KUKA KRL program: MyProgram_130().src

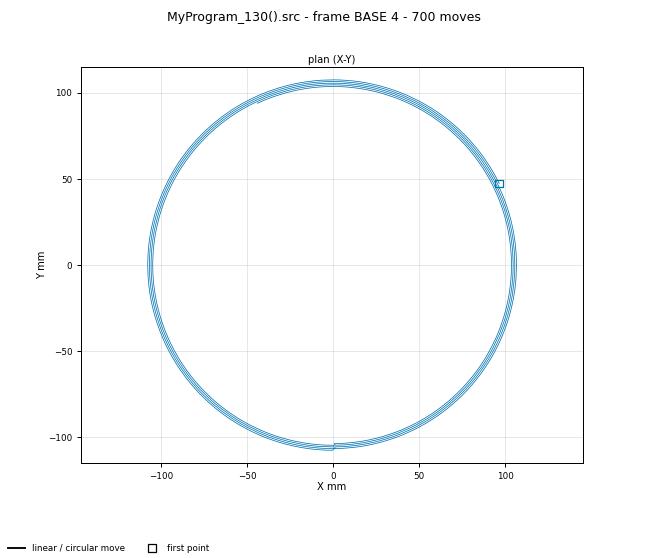
[picture p0: tool path of MyProgram_130().src in frame BASE 4, 700 of 700 moves have a stored position in this frame; points joined in program order, loops and branches not executed]
&ACCESS RVP
&REL 1
&PARAM TEMPLATE = C:\KRC\Roboter\Template\vorgabe
&PARAM EDITMASK = *
DEF MyProgram_130()
; ---- Setting reference (Base) ----
$BASE = BASE_DATA[4]

; --------------------------
; ---- Setting tool (TCP) ----
$TOOL = TOOL_DATA[3]
; --------------------------

$VEL.CP = VEL_APROX_PRINT
Startdeposition()
$VEL.CP = VEL_PRINT
LIN {X 96.6585,Y 47.3768,Z 107,A 22.2478,B 24.9305,C -1.9249,E1 25.1427,E2 423.328} C_DIS
LIN {X 94.8383,Y 50.9225,Z 107,A 24.2361,B 24.9305,C -1.9249,E1 25.1401,E2 421.3499} C_DIS
LIN {X 92.9821,Y 54.2393,Z 107,A 26.2737,B 24.9301,C -1.931,E1 25.1372,E2 419.3085} C_DIS
LIN {X 91.1089,Y 57.3278,Z 107,A 28.1051,B 24.9301,C -1.9322,E1 25.1346,E2 417.4838} C_DIS
LIN {X 89.1092,Y 60.3882,Z 107,A 30.0749,B 24.9296,C -1.9383,E1 25.1315,E2 415.5094} C_DIS
LIN {X 86.9613,Y 63.4425,Z 107,A 31.9479,B 24.9296,C -1.9383,E1 25.1285,E2 413.6455} C_DIS
LIN {X 84.9221,Y 66.1494,Z 107,A 33.8072,B 24.9291,C -1.9451,E1 25.1253,E2 411.779} C_DIS
LIN {X 82.7658,Y 68.826,Z 107,A 35.6176,B 24.9288,C -1.9486,E1 25.1221,E2 409.9685} C_DIS
LIN {X 79.7659,Y 72.2838,Z 107,A 38.1989,B 24.9279,C -1.9604,E1 25.1173,E2 407.3711} C_DIS
LIN {X 76.7784,Y 75.4477,Z 107,A 40.3094,B 24.9282,C -1.9567,E1 25.1132,E2 405.2784} C_DIS
LIN {X 74.3299,Y 77.8622,Z 107,A 42.0113,B 24.9283,C -1.955,E1 25.1098,E2 403.5875} C_DIS
LIN {X 71.8944,Y 80.1149,Z 107,A 43.9014,B 24.9277,C -1.9639,E1 25.1059,E2 401.684} C_DIS
LIN {X 69.2564,Y 82.4081,Z 107,A 45.8045,B 24.9273,C -1.9693,E1 25.1019,E2 399.7755} C_DIS
LIN {X 65.4421,Y 85.4672,Z 107,A 48.451,B 24.9268,C -1.976,E1 25.096,E2 397.1231} C_DIS
LIN {X 62.7263,Y 87.4795,Z 107,A 50.3374,B 24.9263,C -1.9828,E1 25.0918,E2 395.2272} C_DIS
LIN {X 59.7326,Y 89.5519,Z 107,A 52.0715,B 24.9267,C -1.9774,E1 25.0878,E2 393.5119} C_DIS
LIN {X 57.005,Y 91.3106,Z 107,A 53.7544,B 24.9267,C -1.9782,E1 25.0838,E2 391.8323} C_DIS
LIN {X 54.1931,Y 93.0092,Z 107,A 55.7988,B 24.9255,C -1.9932,E1 25.0788,E2 389.7588} C_DIS
LIN {X 50.2355,Y 95.2029,Z 107,A 57.8693,B 24.9263,C -1.9823,E1 25.0738,E2 387.7199} C_DIS
LIN {X 47.8532,Y 96.4223,Z 107,A 59.6078,B 24.9252,C -1.9973,E1 25.0694,E2 385.9507} C_DIS
LIN {X 43.6886,Y 98.3811,Z 107,A 61.7829,B 24.9259,C -1.9886,E1 25.064,E2 383.8015} C_DIS
LIN {X 40.8548,Y 99.59,Z 107,A 63.442,B 24.9257,C -1.9912,E1 25.0597,E2 382.1403} C_DIS
LIN {X 37.0788,Y 101.0564,Z 107,A 65.6254,B 24.9254,C -1.9944,E1 25.054,E2 379.9539} C_DIS
LIN {X 33.3917,Y 102.334,Z 107,A 67.6345,B 24.9254,C -1.9934,E1 25.0487,E2 377.9512} C_DIS
LIN {X 30.598,Y 103.2035,Z 107,A 69.2165,B 24.9254,C -1.9955,E1 25.0444,E2 376.3668} C_DIS
LIN {X 27.4751,Y 104.0802,Z 107,A 71.0057,B 24.9251,C -1.9992,E1 25.0396,E2 374.5718} C_DIS
LIN {X 24.1955,Y 104.8893,Z 107,A 72.6636,B 24.9254,C -1.9945,E1 25.0351,E2 372.9274} C_DIS
LIN {X 19.4871,Y 105.8661,Z 107,A 75.8484,B 24.9234,C -2.0212,E1 25.0262,E2 369.6832} C_DIS
LIN {X 15.5445,Y 106.5163,Z 107,A 77.4337,B 24.925,C -1.9997,E1 25.022,E2 368.1504} C_DIS
LIN {X 12.0252,Y 106.9712,Z 107,A 79.4475,B 24.9246,C -2.0051,E1 25.0164,E2 366.1252} C_DIS
LIN {X 8.1375,Y 107.3367,Z 107,A 81.5895,B 24.9244,C -2.0078,E1 25.0104,E2 363.9779} C_DIS
LIN {X 3.8187,Y 107.5773,Z 107,A 83.6882,B 24.925,C -1.9995,E1 25.0046,E2 361.8996} C_DIS
LIN {X 0.959,Y 107.64,Z 107,A 85.3969,B 24.9245,C -2.0067,E1 24.9998,E2 360.1738} C_DIS
LIN {X -6.6056,Y 107.443,Z 107,A 89.3666,B 24.9248,C -2.0031,E1 24.9887,E2 356.2122} C_DIS
LIN {X -10.3707,Y 107.1442,Z 107,A 92.1892,B 24.9224,C -2.0346,E1 24.9807,E2 353.313} C_DIS
LIN {X -15.902,Y 106.4642,Z 107,A 94.2252,B 24.9253,C -1.9955,E1 24.9753,E2 351.3684} C_DIS
LIN {X -19.0755,Y 105.9402,Z 107,A 95.8763,B 24.9256,C -1.9919,E1 24.9708,E2 349.7242} C_DIS
LIN {X -22.435,Y 105.2812,Z 107,A 97.6602,B 24.9258,C -1.9888,E1 24.9659,E2 347.9455} C_DIS
LIN {X -25.6012,Y 104.5551,Z 107,A 99.5013,B 24.9256,C -1.9916,E1 24.9609,E2 346.0953} C_DIS
LIN {X -28.8893,Y 103.6958,Z 107,A 101.1251,B 24.9263,C -1.9825,E1 24.9566,E2 344.4908} C_DIS
LIN {X -31.4867,Y 102.9366,Z 107,A 102.8288,B 24.9257,C -1.9912,E1 24.9519,E2 342.7635} C_DIS
LIN {X -37.5976,Y 100.8659,Z 107,A 106.2811,B 24.9259,C -1.9875,E1 24.9428,E2 339.3131} C_DIS
LIN {X -41.0114,Y 99.5262,Z 107,A 108.0603,B 24.9266,C -1.9781,E1 24.9383,E2 337.5524} C_DIS
LIN {X -44.3883,Y 98.0658,Z 107,A 110.1145,B 24.9266,C -1.979,E1 24.933,E2 335.4914} C_DIS
LIN {X -48.0689,Y 96.3154,Z 107,A 112.4048,B 24.9265,C -1.9802,E1 24.9272,E2 333.1923} C_DIS
LIN {X -50.9886,Y 94.8024,Z 107,A 114.0879,B 24.9269,C -1.9746,E1 24.9231,E2 331.5177} C_DIS
LIN {X -53.859,Y 93.2012,Z 107,A 115.8714,B 24.927,C -1.9728,E1 24.9188,E2 329.7331} C_DIS
LIN {X -56.3491,Y 91.7183,Z 107,A 117.5087,B 24.927,C -1.9736,E1 24.9149,E2 328.089} C_DIS
LIN {X -59.3917,Y 89.7766,Z 107,A 119.7982,B 24.9262,C -1.984,E1 24.9095,E2 325.7671} C_DIS
LIN {X -62.5149,Y 87.6303,Z 107,A 121.9673,B 24.9261,C -1.9858,E1 24.9045,E2 323.5863} C_DIS
LIN {X -66.0582,Y 84.9921,Z 107,A 123.752,B 24.928,C -1.9591,E1 24.9007,E2 321.8588} C_DIS
LIN {X -69.9051,Y 81.8561,Z 107,A 126.4305,B 24.9284,C -1.9546,E1 24.8949,E2 319.1806} C_DIS
LIN {X -73.3692,Y 78.7658,Z 107,A 129.2092,B 24.9279,C -1.9606,E1 24.8891,E2 316.3765} C_DIS
LIN {X -76.0308,Y 76.2023,Z 107,A 131.5737,B 24.9272,C -1.9709,E1 24.8844,E2 313.9773} C_DIS
LIN {X -79.385,Y 72.6996,Z 107,A 133.1703,B 24.9304,C -1.9272,E1 24.8816,E2 312.4779} C_DIS
LIN {X -83.0404,Y 68.4953,Z 107,A 136.283,B 24.9305,C -1.925,E1 24.8759,E2 309.3563} C_DIS
LIN {X -85.2435,Y 65.7323,Z 107,A 138.1744,B 24.9309,C -1.9204,E1 24.8726,E2 307.467} C_DIS
LIN {X -86.7483,Y 63.7335,Z 107,A 139.524,B 24.9311,C -1.9174,E1 24.8704,E2 306.1179} C_DIS
LIN {X -88.2223,Y 61.6774,Z 107,A 140.9553,B 24.9311,C -1.9169,E1 24.8681,E2 304.6809} C_DIS
LIN {X -89.7399,Y 59.4474,Z 107,A 142.4812,B 24.9311,C -1.9162,E1 24.8657,E2 303.1489} C_DIS
LIN {X -91.7156,Y 56.3535,Z 107,A 144.4514,B 24.9315,C -1.9113,E1 24.8628,E2 301.1806} C_DIS
LIN {X -93.6411,Y 53.0935,Z 107,A 146.4172,B 24.9321,C -1.9036,E1 24.86,E2 299.2228} C_DIS
LIN {X -95.5947,Y 49.4882,Z 107,A 148.929,B 24.9316,C -1.9094,E1 24.8567,E2 296.6836} C_DIS
LIN {X -98.2788,Y 43.9152,Z 107,A 151.9288,B 24.9331,C -1.8886,E1 24.8532,E2 293.7172} C_DIS
LIN {X -99.7804,Y 40.3869,Z 107,A 154.0677,B 24.9333,C -1.886,E1 24.8509,E2 291.5727} C_DIS
LIN {X -101.0566,Y 37.0783,Z 107,A 155.7378,B 24.9343,C -1.8721,E1 24.8493,E2 289.9264} C_DIS
LIN {X -102.2236,Y 33.733,Z 107,A 157.8972,B 24.934,C -1.8763,E1 24.8474,E2 287.7446} C_DIS
LIN {X -103.3972,Y 29.9431,Z 107,A 159.9805,B 24.9345,C -1.8686,E1 24.8457,E2 285.6677} C_DIS
LIN {X -104.3459,Y 26.4433,Z 107,A 162.0668,B 24.9345,C -1.8683,E1 24.8442,E2 283.57} C_DIS
LIN {X -105.411,Y 21.8113,Z 107,A 164.295,B 24.9359,C -1.849,E1 24.8429,E2 281.3746} C_DIS
LIN {X -105.8892,Y 19.3588,Z 107,A 165.5472,B 24.9364,C -1.8418,E1 24.8423,E2 280.1321} C_DIS
LIN {X -106.3948,Y 16.3507,Z 107,A 167.2943,B 24.9364,C -1.8412,E1 24.8415,E2 278.3761} C_DIS
LIN {X -106.8679,Y 12.907,Z 107,A 169.2441,B 24.9366,C -1.8389,E1 24.8408,E2 276.4202} C_DIS
LIN {X -107.1659,Y 10.1354,Z 107,A 171.2847,B 24.9355,C -1.8548,E1 24.8403,E2 274.3293} C_DIS
LIN {X -107.4711,Y 6.0983,Z 107,A 173.0589,B 24.937,C -1.8336,E1 24.84,E2 272.595} C_DIS
LIN {X -107.6446,Y 0.1321,Z 107,A 177.1432,B 24.9353,C -1.8574,E1 24.8398,E2 268.4294} C_DIS
LIN {X -107.4825,Y -5.891,Z 107,A 179.2876,B 24.9388,C -1.8072,E1 24.8401,E2 266.3918} C_DIS
LIN {X -107.2538,Y -9.1743,Z 107,A -178.835,B 24.9388,C -1.8062,E1 24.8405,E2 264.5055} C_DIS
LIN {X -106.9,Y -12.633,Z 107,A -177.0787,B 24.9395,C -1.7968,E1 24.8411,E2 262.761} C_DIS
LIN {X -106.404,Y -16.2911,Z 107,A -175.0871,B 24.9398,C -1.7916,E1 24.8418,E2 260.7701} C_DIS
LIN {X -105.8218,Y -19.7319,Z 107,A -173.144,B 24.94,C -1.7889,E1 24.8428,E2 258.8218} C_DIS
LIN {X -105.1397,Y -23.0837,Z 107,A -171.3092,B 24.9404,C -1.7838,E1 24.8439,E2 256.9885} C_DIS
LIN {X -104.3676,Y -26.3591,Z 107,A -169.601,B 24.9409,C -1.7751,E1 24.845,E2 255.2908} C_DIS
LIN {X -103.6911,Y -28.9061,Z 107,A -168.1051,B 24.9409,C -1.7743,E1 24.8461,E2 253.7882} C_DIS
LIN {X -102.5467,Y -32.7343,Z 107,A -166.2338,B 24.9421,C -1.7584,E1 24.8476,E2 251.9442} C_DIS
LIN {X -100.3685,Y -38.9049,Z 107,A -161.9221,B 24.9407,C -1.7792,E1 24.8518,E2 247.5585} C_DIS
LIN {X -98.8074,Y -42.713,Z 107,A -160.3286,B 24.9426,C -1.7503,E1 24.8535,E2 246.0252} C_DIS
LIN {X -97.4748,Y -45.6719,Z 107,A -158.5346,B 24.9427,C -1.7479,E1 24.8556,E2 244.227} C_DIS
LIN {X -95.6155,Y -49.4482,Z 107,A -155.635,B 24.9415,C -1.7666,E1 24.8594,E2 241.2671} C_DIS
LIN {X -93.4765,Y -53.38,Z 107,A -153.9384,B 24.9436,C -1.7341,E1 24.8616,E2 239.6392} C_DIS
LIN {X -90.6835,Y -57.9976,Z 107,A -151.0601,B 24.9441,C -1.7267,E1 24.8658,E2 236.7638} C_DIS
LIN {X -88.769,Y -60.8908,Z 107,A -149.1874,B 24.9444,C -1.723,E1 24.8687,E2 234.8907} C_DIS
LIN {X -84.9645,Y -66.0944,Z 107,A -145.6186,B 24.9446,C -1.7198,E1 24.8747,E2 231.3124} C_DIS
LIN {X -82.847,Y -68.7282,Z 107,A -143.6718,B 24.9445,C -1.7212,E1 24.8782,E2 229.3531} C_DIS
LIN {X -79.7523,Y -72.2993,Z 107,A -141.2769,B 24.9451,C -1.7108,E1 24.8826,E2 226.9721} C_DIS
LIN {X -77.2011,Y -75.0158,Z 107,A -139.508,B 24.946,C -1.6983,E1 24.886,E2 225.2255} C_DIS
LIN {X -73.4402,Y -78.7014,Z 107,A -136.4935,B 24.9458,C -1.7006,E1 24.8921,E2 222.193} C_DIS
LIN {X -70.9099,Y -80.9876,Z 107,A -134.4839,B 24.9456,C -1.7045,E1 24.8963,E2 220.166} C_DIS
LIN {X -67.7059,Y -83.6846,Z 107,A -132.5306,B 24.9465,C -1.6896,E1 24.9005,E2 218.2408} C_DIS
LIN {X -65.0108,Y -85.7962,Z 107,A -130.1821,B 24.9454,C -1.7069,E1 24.9058,E2 215.8427} C_DIS
LIN {X -61.9127,Y -88.0588,Z 107,A -128.6477,B 24.9469,C -1.6836,E1 24.9092,E2 214.3585} C_DIS
LIN {X -59.5914,Y -89.645,Z 107,A -127.126,B 24.9469,C -1.6821,E1 24.9127,E2 212.8351} C_DIS
LIN {X -57.1592,Y -91.2143,Z 107,A -125.4568,B 24.9469,C -1.6848,E1 24.9167,E2 211.1543} C_DIS
LIN {X -54.2095,Y -92.9997,Z 107,A -123.8481,B 24.9475,C -1.6732,E1 24.9205,E2 209.5683} C_DIS
LIN {X -51.1709,Y -94.7035,Z 107,A -121.5419,B 24.9466,C -1.6886,E1 24.9262,E2 207.2189} C_DIS
LIN {X -48.2988,Y -96.2015,Z 107,A -120.1064,B 24.9474,C -1.6749,E1 24.9297,E2 205.812} C_DIS
LIN {X -45.3758,Y -97.6126,Z 107,A -118.4361,B 24.9477,C -1.6707,E1 24.9339,E2 204.1477} C_DIS
LIN {X -42.3952,Y -98.9457,Z 107,A -116.5495,B 24.9474,C -1.6747,E1 24.9388,E2 202.2471} C_DIS
LIN {X -38.6625,Y -100.4626,Z 107,A -114.4481,B 24.9477,C -1.6709,E1 24.9442,E2 200.1502} C_DIS
LIN {X -34.8861,Y -101.8353,Z 107,A -112.3473,B 24.9479,C -1.6675,E1 24.9498,E2 198.0532} C_DIS
LIN {X -31.6195,Y -102.8955,Z 107,A -110.6303,B 24.9483,C -1.6617,E1 24.9543,E2 196.347} C_DIS
LIN {X -28.2364,Y -103.8746,Z 107,A -108.7476,B 24.9483,C -1.6608,E1 24.9594,E2 194.4634} C_DIS
LIN {X -22.766,Y -105.209,Z 107,A -105.0637,B 24.9467,C -1.6871,E1 24.9696,E2 190.7123} C_DIS
LIN {X -18.4933,Y -106.0449,Z 107,A -103.4736,B 24.9486,C -1.6567,E1 24.9738,E2 189.1928} C_DIS
LIN {X -14.0235,Y -106.7266,Z 107,A -100.9849,B 24.9484,C -1.6594,E1 24.9807,E2 186.6955} C_DIS
LIN {X -11.0399,Y -107.0763,Z 107,A -99.303,B 24.9482,C -1.6626,E1 24.9854,E2 185.0049} C_DIS
LIN {X -7.2203,Y -107.4014,Z 107,A -97.2958,B 24.9482,C -1.6613,E1 24.9909,E2 183.0002} C_DIS
LIN {X -4.2877,Y -107.5589,Z 107,A -95.7906,B 24.9484,C -1.659,E1 24.9951,E2 181.5} C_DIS
LIN {X -0.1666,Y -107.6448,Z 107,A -93.638,B 24.9485,C -1.6577,E1 25.0011,E2 179.3504} C_DIS
LIN {X -0.1666,Y -107.6448,Z 107,A -93.638,B 24.9485,C -1.6577,E1 25.0011,E2 179.3504} C_DIS
Enddeposition()
LIN {X 0.7291,Y -106.6759,Z 107,A -92.7811,B 24.9465,C -1.6901,E1 25.0037,E2 178.4168} C_DIS
Startdeposition()
$VEL.CP = VEL_PRINT
LIN {X -4.5777,Y -106.5805,Z 107,A -96.6006,B 24.949,C -1.6502,E1 24.9928,E2 182.331} C_DIS
LIN {X -7.3432,Y -106.4259,Z 107,A -98.8577,B 24.9508,C -1.6196,E1 24.9863,E2 184.6615} C_DIS
LIN {X -11.3426,Y -106.0743,Z 107,A -100.5047,B 24.9496,C -1.6399,E1 24.9819,E2 186.2613} C_DIS
LIN {X -16.3427,Y -105.4196,Z 107,A -103.0853,B 24.9493,C -1.6456,E1 24.9748,E2 188.8305} C_DIS
LIN {X -20.2997,Y -104.7297,Z 107,A -105.6247,B 24.9501,C -1.6313,E1 24.9677,E2 191.4064} C_DIS
LIN {X -25.2157,Y -103.6558,Z 107,A -108.0224,B 24.9493,C -1.6446,E1 24.9612,E2 193.7756} C_DIS
LIN {X -28.5439,Y -102.7907,Z 107,A -109.9612,B 24.9495,C -1.6421,E1 24.956,E2 195.7232} C_DIS
LIN {X -32.2364,Y -101.6936,Z 107,A -112.0458,B 24.9495,C -1.643,E1 24.9504,E2 197.8093} C_DIS
LIN {X -35.7308,Y -100.518,Z 107,A -114.0608,B 24.9494,C -1.6433,E1 24.9451,E2 199.8275} C_DIS
LIN {X -39.5817,Y -99.0658,Z 107,A -116.7004,B 24.9503,C -1.629,E1 24.9381,E2 202.507} C_DIS
LIN {X -43.2409,Y -97.5244,Z 107,A -119.7156,B 24.9522,C -1.598,E1 24.9303,E2 205.6032} C_DIS
LIN {X -49.9658,Y -94.2542,Z 107,A -122.2311,B 24.9484,C -1.6599,E1 24.9244,E2 207.9782} C_DIS
LIN {X -53.1252,Y -92.5099,Z 107,A -124.2107,B 24.9483,C -1.661,E1 24.9195,E2 209.9609} C_DIS
LIN {X -57.943,Y -89.5718,Z 107,A -127.1853,B 24.9479,C -1.6677,E1 24.9125,E2 212.9289} C_DIS
LIN {X -64.0498,Y -85.3111,Z 107,A -130.9543,B 24.9469,C -1.6832,E1 24.9039,E2 216.6741} C_DIS
LIN {X -66.0683,Y -83.7577,Z 107,A -132.705,B 24.9477,C -1.6711,E1 24.9,E2 218.4599} C_DIS
LIN {X -70.1053,Y -80.409,Z 107,A -135.1368,B 24.9464,C -1.691,E1 24.8949,E2 220.8536} C_DIS
LIN {X -72.1428,Y -78.5861,Z 107,A -137.9367,B 24.9493,C -1.6443,E1 24.8889,E2 223.7762} C_DIS
LIN {X -76.1514,Y -74.7092,Z 107,A -139.7878,B 24.9463,C -1.6931,E1 24.8854,E2 225.5188} C_DIS
LIN {X -77.9434,Y -72.8376,Z 107,A -141.4089,B 24.9466,C -1.6875,E1 24.8822,E2 227.1602} C_DIS
LIN {X -81.2627,Y -69.114,Z 107,A -144.0627,B 24.9462,C -1.6946,E1 24.8774,E2 229.8092} C_DIS
LIN {X -83.844,Y -65.9584,Z 107,A -147.1595,B 24.948,C -1.6665,E1 24.8719,E2 232.9876} C_DIS
LIN {X -86.9878,Y -61.7539,Z 107,A -149.0102,B 24.9453,C -1.709,E1 24.869,E2 234.7459} C_DIS
LIN {X -88.4889,Y -59.5831,Z 107,A -150.5347,B 24.9453,C -1.7087,E1 24.8666,E2 236.2787} C_DIS
LIN {X -91.0172,Y -55.6444,Z 107,A -152.812,B 24.9443,C -1.724,E1 24.8632,E2 238.5311} C_DIS
LIN {X -92.4216,Y -53.2788,Z 107,A -155.2985,B 24.9464,C -1.691,E1 24.8596,E2 241.1091} C_DIS
LIN {X -94.7068,Y -49.1058,Z 107,A -157.0324,B 24.944,C -1.728,E1 24.8574,E2 242.7642} C_DIS
LIN {X -96.0703,Y -46.3778,Z 107,A -158.8272,B 24.9441,C -1.7268,E1 24.8552,E2 244.5714} C_DIS
LIN {X -97.713,Y -42.8085,Z 107,A -161.0908,B 24.9441,C -1.7273,E1 24.8526,E2 246.8464} C_DIS
LIN {X -99.12,Y -39.4438,Z 107,A -162.6893,B 24.9429,C -1.7461,E1 24.8509,E2 248.4089} C_DIS
LIN {X -100.1706,Y -36.6911,Z 107,A -164.9697,B 24.9442,C -1.7254,E1 24.8487,E2 250.7514} C_DIS
LIN {X -101.3987,Y -33.1477,Z 107,A -166.3239,B 24.9422,C -1.7554,E1 24.8475,E2 252.0419} C_DIS
LIN {X -102.3933,Y -29.9359,Z 107,A -168.0463,B 24.9417,C -1.7639,E1 24.8461,E2 253.754} C_DIS
LIN {X -103.3792,Y -26.328,Z 107,A -170.2868,B 24.9418,C -1.7616,E1 24.8445,E2 256.013} C_DIS
LIN {X -104.222,Y -22.7627,Z 107,A -172.2967,B 24.9415,C -1.7662,E1 24.8432,E2 258.0237} C_DIS
LIN {X -104.9138,Y -19.3302,Z 107,A -174.2434,B 24.9413,C -1.7697,E1 24.8422,E2 259.9736} C_DIS
LIN {X -105.5055,Y -15.787,Z 107,A -176.2606,B 24.9411,C -1.7726,E1 24.8413,E2 261.9959} C_DIS
LIN {X -105.9819,Y -12.1756,Z 107,A -178.0179,B 24.9402,C -1.786,E1 24.8407,E2 263.7317} C_DIS
LIN {X -106.2865,Y -9.1625,Z 107,A -179.877,B 24.9404,C -1.7828,E1 24.8403,E2 265.6096} C_DIS
LIN {X -106.5453,Y -5.3608,Z 107,A 177.4172,B 24.9416,C -1.7658,E1 24.8399,E2 268.3722} C_DIS
LIN {X -106.6767,Y -0.652,Z 107,A 175.6237,B 24.9393,C -1.8003,E1 24.8398,E2 270.0941} C_DIS
LIN {X -106.5914,Y 4.3116,Z 107,A 172.6262,B 24.9395,C -1.7971,E1 24.84,E2 273.1175} C_DIS
LIN {X -106.2677,Y 9.3669,Z 107,A 170.4075,B 24.9376,C -1.8239,E1 24.8405,E2 275.2855} C_DIS
LIN {X -105.9316,Y 12.6055,Z 107,A 168.3992,B 24.9379,C -1.8202,E1 24.8411,E2 277.3147} C_DIS
LIN {X -105.4294,Y 16.2789,Z 107,A 166.4301,B 24.9374,C -1.8274,E1 24.8419,E2 279.2783} C_DIS
LIN {X -104.7835,Y 20.0199,Z 107,A 164.4335,B 24.9368,C -1.8355,E1 24.8429,E2 281.2675} C_DIS
LIN {X -104.1067,Y 23.2913,Z 107,A 161.8248,B 24.9385,C -1.8121,E1 24.8445,E2 283.9472} C_DIS
LIN {X -102.9858,Y 27.826,Z 107,A 160.2332,B 24.9356,C -1.8529,E1 24.8456,E2 285.4509} C_DIS
LIN {X -102.2242,Y 30.5057,Z 107,A 158.5898,B 24.9356,C -1.8523,E1 24.8468,E2 287.1051} C_DIS
LIN {X -100.3189,Y 36.2844,Z 107,A 154.3083,B 24.9375,C -1.8263,E1 24.8508,E2 291.4731} C_DIS
LIN {X -98.3135,Y 41.4104,Z 107,A 152.2794,B 24.9346,C -1.8685,E1 24.8529,E2 293.4126} C_DIS
LIN {X -96.3866,Y 45.718,Z 107,A 149.5924,B 24.9344,C -1.8706,E1 24.856,E2 296.1092} C_DIS
LIN {X -93.6934,Y 51.0093,Z 107,A 147.0183,B 24.9322,C -1.9024,E1 24.8592,E2 298.6214} C_DIS
LIN {X -92.54,Y 53.0727,Z 107,A 145.2101,B 24.9333,C -1.8865,E1 24.8618,E2 300.477} C_DIS
LIN {X -90.6367,Y 56.2622,Z 107,A 142.9746,B 24.9335,C -1.8835,E1 24.8651,E2 302.7311} C_DIS
LIN {X -88.2571,Y 59.9255,Z 107,A 140.9093,B 24.9323,C -1.9002,E1 24.8682,E2 304.7668} C_DIS
LIN {X -86.2594,Y 62.7676,Z 107,A 139.009,B 24.932,C -1.9041,E1 24.8713,E2 306.6672} C_DIS
LIN {X -84.2742,Y 65.4092,Z 107,A 137.1172,B 24.932,C -1.9046,E1 24.8745,E2 308.5667} C_DIS
LIN {X -81.9514,Y 68.296,Z 107,A 135.0118,B 24.932,C -1.9056,E1 24.8782,E2 310.6794} C_DIS
LIN {X -78.2741,Y 72.4829,Z 107,A 131.8307,B 24.9319,C -1.9064,E1 24.8842,E2 313.873} C_DIS
LIN {X -74.4759,Y 76.3812,Z 107,A 128.533,B 24.9323,C -1.8998,E1 24.8908,E2 317.2002} C_DIS
LIN {X -71.1501,Y 79.486,Z 107,A 126.2097,B 24.9316,C -1.9098,E1 24.8956,E2 319.509} C_DIS
LIN {X -68.04,Y 82.1642,Z 107,A 124.713,B 24.9294,C -1.9407,E1 24.8987,E2 320.9379} C_DIS
LIN {X -65.7851,Y 83.9816,Z 107,A 122.5971,B 24.9306,C -1.9234,E1 24.9034,E2 323.1028} C_DIS
LIN {X -63.1014,Y 86.015,Z 107,A 121.0445,B 24.9297,C -1.9366,E1 24.9068,E2 324.6295} C_DIS
LIN {X -59.556,Y 88.5073,Z 107,A 118.7864,B 24.9292,C -1.9438,E1 24.912,E2 326.8781} C_DIS
LIN {X -54.5917,Y 91.6528,Z 107,A 115.6118,B 24.9288,C -1.949,E1 24.9196,E2 330.0503} C_DIS
LIN {X -51.1585,Y 93.6124,Z 107,A 113.5901,B 24.9282,C -1.9565,E1 24.9244,E2 332.06} C_DIS
LIN {X -48.2699,Y 95.134,Z 107,A 111.7593,B 24.9282,C -1.9565,E1 24.929,E2 333.8957} C_DIS
LIN {X -44.5289,Y 96.9424,Z 107,A 109.0327,B 24.9293,C -1.9415,E1 24.936,E2 336.665} C_DIS
LIN {X -40.9976,Y 98.4874,Z 107,A 107.5941,B 24.9274,C -1.9681,E1 24.9396,E2 338.0435} C_DIS
LIN {X -33.9765,Y 101.1236,Z 107,A 103.5054,B 24.9272,C -1.971,E1 24.9503,E2 342.1335} C_DIS
LIN {X -29.3258,Y 102.5691,Z 107,A 101.0121,B 24.9266,C -1.9786,E1 24.9569,E2 344.6131} C_DIS
LIN {X -26.1082,Y 103.4357,Z 107,A 99.1217,B 24.9267,C -1.9766,E1 24.962,E2 346.5113} C_DIS
LIN {X -23.4946,Y 104.0608,Z 107,A 97.4027,B 24.9274,C -1.9674,E1 24.9668,E2 348.2544} C_DIS
LIN {X -19.5268,Y 104.8785,Z 107,A 95.3081,B 24.9271,C -1.9722,E1 24.9725,E2 350.3397} C_DIS
LIN {X -16.0378,Y 105.4667,Z 107,A 92.8306,B 24.9286,C -1.9515,E1 24.9795,E2 352.8686} C_DIS
LIN {X -11.5923,Y 106.0482,Z 107,A 91.0619,B 24.9267,C -1.9773,E1 24.9842,E2 354.5771} C_DIS
LIN {X -8.7774,Y 106.3174,Z 107,A 88.6684,B 24.9291,C -1.9444,E1 24.9911,E2 357.0497} C_DIS
LIN {X -3.4124,Y 106.6243,Z 107,A 85.8592,B 24.9288,C -1.9483,E1 24.9989,E2 359.8503} C_DIS
LIN {X 1.6641,Y 106.6662,Z 107,A 84.1246,B 24.926,C -1.9872,E1 25.0035,E2 361.4924} C_DIS
LIN {X 5.8471,Y 106.5184,Z 107,A 81.6319,B 24.9267,C -1.9777,E1 25.0105,E2 364.0068} C_DIS
LIN {X 12.6533,Y 105.926,Z 107,A 77.9766,B 24.9267,C -1.9779,E1 25.0207,E2 367.6596} C_DIS
LIN {X 17.7317,Y 105.1949,Z 107,A 75.1933,B 24.9267,C -1.976,E1 25.0283,E2 370.4448} C_DIS
LIN {X 21.5402,Y 104.4815,Z 107,A 73.3282,B 24.9262,C -1.9836,E1 25.0334,E2 372.2894} C_DIS
LIN {X 24.2404,Y 103.8885,Z 107,A 71.8289,B 24.9263,C -1.9823,E1 25.0375,E2 373.7899} C_DIS
LIN {X 26.7324,Y 103.2752,Z 107,A 70.3354,B 24.9267,C -1.9769,E1 25.0415,E2 375.2941} C_DIS
LIN {X 30.3254,Y 102.2777,Z 107,A 68.335,B 24.9268,C -1.9756,E1 25.0469,E2 377.2941} C_DIS
LIN {X 34.773,Y 100.8541,Z 107,A 65.8701,B 24.9268,C -1.9752,E1 25.0534,E2 379.7552} C_DIS
LIN {X 39.9525,Y 98.9153,Z 107,A 62.886,B 24.9271,C -1.9718,E1 25.0612,E2 382.7409} C_DIS
LIN {X 46.6383,Y 95.9451,Z 107,A 59.256,B 24.9265,C -1.9794,E1 25.0704,E2 386.344} C_DIS
LIN {X 49.8773,Y 94.3009,Z 107,A 57.069,B 24.9274,C -1.9672,E1 25.0759,E2 388.5537} C_DIS
LIN {X 54.6412,Y 91.6236,Z 107,A 54.1977,B 24.9276,C -1.9656,E1 25.0829,E2 391.4202} C_DIS
LIN {X 57.2818,Y 89.9962,Z 107,A 51.5658,B 24.9306,C -1.9237,E1 25.0893,E2 394.1427} C_DIS
LIN {X 61.6176,Y 87.0851,Z 107,A 49.8426,B 24.9277,C -1.9631,E1 25.093,E2 395.7668} C_DIS
LIN {X 64.7101,Y 84.8129,Z 107,A 46.988,B 24.9304,C -1.9269,E1 25.0995,E2 398.6968} C_DIS
LIN {X 67.9092,Y 82.2729,Z 107,A 45.6373,B 24.9282,C -1.9575,E1 25.1023,E2 399.9701} C_DIS
LIN {X 70.0114,Y 80.4911,Z 107,A 43.205,B 24.9312,C -1.9153,E1 25.1076,E2 402.4926} C_DIS
LIN {X 73.4728,Y 77.3459,Z 107,A 41.4831,B 24.9292,C -1.9427,E1 25.111,E2 404.1426} C_DIS
LIN {X 75.8206,Y 75.044,Z 107,A 39.6793,B 24.9296,C -1.9373,E1 25.1146,E2 405.9515} C_DIS
LIN {X 79.7841,Y 70.8171,Z 107,A 36.722,B 24.9296,C -1.9368,E1 25.1202,E2 408.8969} C_DIS
LIN {X 81.3388,Y 69.0247,Z 107,A 35.2285,B 24.9306,C -1.9247,E1 25.1229,E2 410.4124} C_DIS
LIN {X 84.8257,Y 64.6935,Z 107,A 32.4554,B 24.9304,C -1.9264,E1 25.1277,E2 413.1683} C_DIS
LIN {X 86.2615,Y 62.7648,Z 107,A 31.11,B 24.9308,C -1.921,E1 25.1299,E2 414.5202} C_DIS
LIN {X 89.2777,Y 58.3953,Z 107,A 28.5202,B 24.9305,C -1.9247,E1 25.134,E2 417.0883} C_DIS
LIN {X 91.277,Y 55.2171,Z 107,A 26.2521,B 24.9317,C -1.9088,E1 25.1374,E2 419.3827} C_DIS
LIN {X 93.7671,Y 50.8733,Z 107,A 23.9359,B 24.9311,C -1.9173,E1 25.1405,E2 421.6666} C_DIS
LIN {X 94.9283,Y 48.6725,Z 107,A 21.689,B 24.9341,C -1.875,E1 25.1435,E2 424.0015} C_DIS
LIN {X 96.601,Y 45.2625,Z 107,A 20.4535,B 24.9321,C -1.9033,E1 25.1449,E2 425.1635} C_DIS
LIN {X 97.6788,Y 42.887,Z 107,A 18.7521,B 24.9333,C -1.8865,E1 25.1469,E2 426.8954} C_DIS
LIN {X 99.0774,Y 39.5522,Z 107,A 16.8115,B 24.9337,C -1.8809,E1 25.1489,E2 428.8386} C_DIS
LIN {X 100.7645,Y 35.0282,Z 107,A 14.4192,B 24.9337,C -1.8818,E1 25.1512,E2 431.2154} C_DIS
LIN {X 101.5484,Y 32.6851,Z 107,A 12.9356,B 24.9344,C -1.8711,E1 25.1525,E2 432.7158} C_DIS
LIN {X 102.5993,Y 29.2193,Z 107,A 11.067,B 24.9346,C -1.8684,E1 25.154,E2 434.5799} C_DIS
LIN {X 103.4362,Y 26.105,Z 107,A 9.4367,B 24.9346,C -1.8674,E1 25.1551,E2 436.2031} C_DIS
LIN {X 104.1092,Y 23.2798,Z 107,A 7.0936,B 24.9373,C -1.8292,E1 25.1566,E2 438.623} C_DIS
LIN {X 104.966,Y 19.04,Z 107,A 5.2432,B 24.9364,C -1.842,E1 25.1576,E2 440.4323} C_DIS
LIN {X 105.8398,Y 13.3575,Z 107,A 1.3285,B 24.9395,C -1.7971,E1 25.159,E2 444.4298} C_DIS
LIN {X 106.4215,Y 7.4082,Z 107,A -0.5743,B 24.9364,C -1.8426,E1 25.1594,E2 446.2141} C_DIS
LIN {X 106.6395,Y 2.9158,Z 107,A -3.2478,B 24.9377,C -1.8236,E1 25.1598,E2 448.9164} C_DIS
LIN {X 106.6758,Y -0.8204,Z 107,A -5.4825,B 24.9388,C -1.8073,E1 25.1598,E2 451.1761} C_DIS
LIN {X 106.3917,Y -7.8464,Z 107,A -8.899,B 24.9386,C -1.8106,E1 25.1593,E2 454.5648} C_DIS
LIN {X 106.1076,Y -11.0245,Z 107,A -10.6212,B 24.939,C -1.8047,E1 25.1588,E2 456.2907} C_DIS
LIN {X 105.7358,Y -14.16,Z 107,A -12.2459,B 24.9391,C -1.8022,E1 25.1583,E2 457.9115} C_DIS
LIN {X 104.9214,Y -19.2882,Z 107,A -15.1436,B 24.94,C -1.7885,E1 25.1569,E2 460.8245} C_DIS
LIN {X 104.221,Y -22.7673,Z 107,A -17.1882,B 24.9409,C -1.7764,E1 25.1557,E2 462.8857} C_DIS
LIN {X 102.9844,Y -27.831,Z 107,A -19.6651,B 24.9405,C -1.7814,E1 25.1541,E2 465.3366} C_DIS
LIN {X 102.174,Y -30.675,Z 107,A -21.3296,B 24.9411,C -1.7731,E1 25.1527,E2 467.0113} C_DIS
LIN {X 100.9401,Y -34.5205,Z 107,A -23.3686,B 24.9411,C -1.7718,E1 25.151,E2 469.0416} C_DIS
LIN {X 99.3396,Y -38.8848,Z 107,A -25.9866,B 24.942,C -1.7588,E1 25.1484,E2 471.6756} C_DIS
LIN {X 97.9855,Y -42.1834,Z 107,A -27.9605,B 24.9426,C -1.7504,E1 25.1463,E2 473.6585} C_DIS
LIN {X 96.5101,Y -45.4577,Z 107,A -29.7403,B 24.9426,C -1.751,E1 25.1442,E2 475.4274} C_DIS
LIN {X 94.3938,Y -49.7008,Z 107,A -32.2374,B 24.9429,C -1.7455,E1 25.1411,E2 477.9242} C_DIS
LIN {X 93.1411,Y -52.0105,Z 107,A -33.7023,B 24.9433,C -1.739,E1 25.1391,E2 479.3967} C_DIS
LIN {X 91.4761,Y -54.8894,Z 107,A -35.8656,B 24.9447,C -1.7177,E1 25.1359,E2 481.5991} C_DIS
LIN {X 89.1785,Y -58.5457,Z 107,A -37.7537,B 24.9439,C -1.7295,E1 25.1331,E2 483.4499} C_DIS
LIN {X 85.9776,Y -63.1525,Z 107,A -40.7401,B 24.9444,C -1.7223,E1 25.1284,E2 486.4388} C_DIS
LIN {X 82.5496,Y -67.5736,Z 107,A -43.6897,B 24.9448,C -1.7165,E1 25.1233,E2 489.3882} C_DIS
LIN {X 80.6317,Y -69.8504,Z 107,A -45.9558,B 24.9469,C -1.6841,E1 25.119,E2 491.7206} C_DIS
LIN {X 77.9814,Y -72.7971,Z 107,A -47.8368,B 24.9465,C -1.6891,E1 25.1155,E2 493.5813} C_DIS
LIN {X 74.7402,Y -76.1207,Z 107,A -50.0337,B 24.9461,C -1.6955,E1 25.1112,E2 495.7537} C_DIS
LIN {X 71.9776,Y -78.7378,Z 107,A -52.3408,B 24.9471,C -1.6796,E1 25.1064,E2 498.0892} C_DIS
LIN {X 67.0116,Y -83.0051,Z 107,A -55.5848,B 24.9469,C -1.6831,E1 25.0995,E2 501.3122} C_DIS
LIN {X 64.0846,Y -85.285,Z 107,A -57.5507,B 24.9471,C -1.68,E1 25.0951,E2 503.2784} C_DIS
LIN {X 60.1953,Y -88.0743,Z 107,A -60.1964,B 24.9476,C -1.6715,E1 25.0891,E2 505.9349} C_DIS
LIN {X 56.729,Y -90.3451,Z 107,A -62.0982,B 24.9471,C -1.6808,E1 25.0847,E2 507.8086} C_DIS
LIN {X 53.6915,Y -92.1834,Z 107,A -64.806,B 24.9494,C -1.6439,E1 25.078,E2 510.5954} C_DIS
LIN {X 50.022,Y -94.2246,Z 107,A -66.5396,B 24.9483,C -1.6616,E1 25.0738,E2 512.2822} C_DIS
LIN {X 47.2373,Y -95.6505,Z 107,A -68.1612,B 24.9483,C -1.6613,E1 25.0698,E2 513.9002} C_DIS
LIN {X 41.4044,Y -98.316,Z 107,A -71.1174,B 24.9473,C -1.6762,E1 25.0624,E2 516.8136} C_DIS
LIN {X 39.5268,Y -99.0874,Z 107,A -72.7329,B 24.9488,C -1.6529,E1 25.0581,E2 518.4807} C_DIS
LIN {X 35.9658,Y -100.4351,Z 107,A -74.8165,B 24.9491,C -1.6485,E1 25.0526,E2 520.5702} C_DIS
LIN {X 30.556,Y -102.2093,Z 107,A -77.4159,B 24.9481,C -1.6637,E1 25.0458,E2 523.1288} C_DIS
LIN {X 27.118,Y -103.1761,Z 107,A -79.7138,B 24.9492,C -1.646,E1 25.0395,E2 525.4649} C_DIS
LIN {X 23.7247,Y -104.0076,Z 107,A -81.4376,B 24.949,C -1.6505,E1 25.0348,E2 527.1758} C_DIS
LIN {X 19.9918,Y -104.7888,Z 107,A -83.4926,B 24.949,C -1.6484,E1 25.0292,E2 529.2331} C_DIS
LIN {X 16.0829,Y -105.4597,Z 107,A -86.4013,B 24.9511,C -1.6154,E1 25.021,E2 532.2172} C_DIS
LIN {X 11.46,Y -106.062,Z 107,A -88.3864,B 24.9499,C -1.6347,E1 25.0156,E2 534.155} C_DIS
LIN {X 5.6821,Y -106.5275,Z 107,A -91.2475,B 24.9494,C -1.6434,E1 25.0077,E2 536.9942} C_DIS
LIN {X 0.7291,Y -106.6759,Z 107,A -92.7773,B 24.9466,C -1.6885,E1 25.0038,E2 538.4168} C_DIS
Enddeposition()
LIN {X 0.7291,Y -106.6759,Z 107,A -92.7773,B 24.9466,C -1.6885,E1 25.0038,E2 538.4168} C_DIS
Startdeposition()
$VEL.CP = VEL_PRINT
LIN {X 1.2934,Y -105.7078,Z 107,A -92.1572,B 24.9447,C -1.7179,E1 25.0057,E2 537.7272} C_DIS
LIN {X 5.6649,Y -105.562,Z 107,A -90.5684,B 24.9467,C -1.687,E1 25.0099,E2 536.2122} C_DIS
LIN {X 10.7499,Y -105.1661,Z 107,A -87.7251,B 24.9464,C -1.6916,E1 25.0178,E2 533.3595} C_DIS
LIN {X 15.8483,Y -104.5195,Z 107,A -84.9135,B 24.9462,C -1.6944,E1 25.0256,E2 530.5435} C_DIS
LIN {X 19.1788,Y -103.9605,Z 107,A -83.3157,B 24.9467,C -1.6864,E1 25.0299,E2 528.9665} C_DIS
LIN {X 22.7586,Y -103.2352,Z 107,A -81.0442,B 24.9458,C -1.7001,E1 25.0362,E2 526.6654} C_DIS
LIN {X 26.3227,Y -102.3841,Z 107,A -79.1377,B 24.9459,C -1.6988,E1 25.0414,E2 524.7647} C_DIS
LIN {X 30.7088,Y -101.1571,Z 107,A -75.7599,B 24.9433,C -1.7395,E1 25.0507,E2 521.2965} C_DIS
LIN {X 35.8261,Y -99.4589,Z 107,A -73.7581,B 24.9455,C -1.7048,E1 25.0557,E2 519.3809} C_DIS
LIN {X 39.4143,Y -98.0925,Z 107,A -70.5639,B 24.9423,C -1.7545,E1 25.0643,E2 516.0764} C_DIS
LIN {X 45.1877,Y -95.5713,Z 107,A -68.1916,B 24.9448,C -1.7158,E1 25.07,E2 513.8016} C_DIS
LIN {X 48.3235,Y -94.0228,Z 107,A -65.3157,B 24.9419,C -1.7605,E1 25.0774,E2 510.828} C_DIS
LIN {X 53.6566,Y -91.0845,Z 107,A -63.1229,B 24.9446,C -1.7195,E1 25.0825,E2 508.7387} C_DIS
LIN {X 56.5463,Y -89.3212,Z 107,A -61.3898,B 24.9446,C -1.7187,E1 25.0866,E2 507.013} C_DIS
LIN {X 60.3529,Y -86.7924,Z 107,A -58.4164,B 24.943,C -1.7447,E1 25.0935,E2 503.9882} C_DIS
LIN {X 63.1083,Y -84.8114,Z 107,A -56.8965,B 24.9436,C -1.735,E1 25.0969,E2 502.4967} C_DIS
LIN {X 67.1642,Y -81.6366,Z 107,A -54.0461,B 24.943,C -1.7436,E1 25.1031,E2 499.6366} C_DIS
LIN {X 72.5204,Y -76.9169,Z 107,A -50.3187,B 24.9428,C -1.7466,E1 25.1109,E2 495.9171} C_DIS
LIN {X 77.2731,Y -72.1416,Z 107,A -46.5034,B 24.9418,C -1.7626,E1 25.1183,E2 492.0804} C_DIS
LIN {X 81.0634,Y -67.8547,Z 107,A -43.1639,B 24.9406,C -1.7809,E1 25.1244,E2 488.7129} C_DIS
LIN {X 83.3051,Y -65.0813,Z 107,A -41.5293,B 24.9411,C -1.7732,E1 25.1272,E2 487.104} C_DIS
LIN {X 85.979,Y -61.5063,Z 107,A -39.1716,B 24.9408,C -1.7772,E1 25.1311,E2 484.7482} C_DIS
LIN {X 88.3339,Y -58.0735,Z 107,A -37.1485,B 24.941,C -1.7735,E1 25.1342,E2 482.7439} C_DIS
LIN {X 90.7843,Y -54.1646,Z 107,A -34.5532,B 24.9403,C -1.7848,E1 25.138,E2 480.1352} C_DIS
LIN {X 92.4394,Y -51.2878,Z 107,A -32.866,B 24.9403,C -1.7852,E1 25.1403,E2 478.4556} C_DIS
LIN {X 93.7805,Y -48.7943,Z 107,A -30.2198,B 24.9367,C -1.8381,E1 25.1439,E2 475.6987} C_DIS
LIN {X 96.3699,Y -43.454,Z 107,A -28.0983,B 24.9393,C -1.8001,E1 25.1462,E2 473.6783} C_DIS
LIN {X 97.5834,Y -40.6578,Z 107,A -25.4381,B 24.9359,C -1.8491,E1 25.1492,E2 470.9173} C_DIS
LIN {X 99.646,Y -35.3011,Z 107,A -23.6056,B 24.9391,C -1.8031,E1 25.1508,E2 469.2034} C_DIS
LIN {X 100.8518,Y -31.6936,Z 107,A -21.3213,B 24.938,C -1.8192,E1 25.1528,E2 466.8941} C_DIS
LIN {X 101.7033,Y -28.8416,Z 107,A -19.9471,B 24.9383,C -1.814,E1 25.1539,E2 465.54} C_DIS
LIN {X 102.8572,Y -24.4171,Z 107,A -17.2016,B 24.937,C -1.8334,E1 25.1558,E2 462.7646} C_DIS
LIN {X 103.5806,Y -21.1298,Z 107,A -15.4494,B 24.9368,C -1.8362,E1 25.1568,E2 461.0162} C_DIS
LIN {X 104.2243,Y -17.685,Z 107,A -13.2879,B 24.9356,C -1.8537,E1 25.1579,E2 458.826} C_DIS
LIN {X 105.2181,Y -10.2379,Z 107,A -9.4638,B 24.9354,C -1.856,E1 25.1592,E2 455.019} C_DIS
LIN {X 105.6236,Y -4.3683,Z 107,A -5.6865,B 24.9329,C -1.892,E1 25.1598,E2 451.1793} C_DIS
LIN {X 105.7151,Y -0.0204,Z 107,A -3.9107,B 24.9341,C -1.8743,E1 25.1598,E2 449.4559} C_DIS
LIN {X 105.4739,Y 7.1174,Z 107,A -0.3852,B 24.9343,C -1.8718,E1 25.1594,E2 445.9571} C_DIS
LIN {X 105.0036,Y 12.2331,Z 107,A 2.5992,B 24.9331,C -1.8893,E1 25.1586,E2 442.9491} C_DIS
LIN {X 104.6404,Y 15.027,Z 107,A 4.7749,B 24.9307,C -1.9223,E1 25.1577,E2 440.7085} C_DIS
LIN {X 103.9397,Y 19.2928,Z 107,A 6.8787,B 24.9309,C -1.9192,E1 25.1566,E2 438.6243} C_DIS
LIN {X 103.293,Y 22.4932,Z 107,A 8.208,B 24.9319,C -1.9057,E1 25.1559,E2 437.3345} C_DIS
LIN {X 102.5532,Y 25.6633,Z 107,A 10.124,B 24.9311,C -1.9177,E1 25.1546,E2 435.4013} C_DIS
LIN {X 101.4994,Y 29.5559,Z 107,A 12.2886,B 24.9306,C -1.9235,E1 25.1529,E2 433.2356} C_DIS
LIN {X 100.3709,Y 33.1883,Z 107,A 14.2737,B 24.9304,C -1.9264,E1 25.1512,E2 431.2548} C_DIS
LIN {X 98.1584,Y 39.2522,Z 107,A 17.7582,B 24.9297,C -1.9361,E1 25.1478,E2 427.7669} C_DIS
LIN {X 95.8522,Y 44.5842,Z 107,A 21.1883,B 24.9282,C -1.9572,E1 25.1439,E2 424.3056} C_DIS
LIN {X 94.3962,Y 47.5929,Z 107,A 22.7428,B 24.9286,C -1.9512,E1 25.142,E2 422.7735} C_DIS
LIN {X 92.6959,Y 50.8242,Z 107,A 25.3675,B 24.9262,C -1.9844,E1 25.1384,E2 420.0842} C_DIS
LIN {X 90.2548,Y 55.0409,Z 107,A 27.1393,B 24.9284,C -1.9542,E1 25.1359,E2 418.3926} C_DIS
LIN {X 86.505,Y 60.7663,Z 107,A 30.9441,B 24.9274,C -1.9678,E1 25.13,E2 414.5748} C_DIS
LIN {X 84.4475,Y 63.5927,Z 107,A 32.6678,B 24.9276,C -1.9652,E1 25.1272,E2 412.8653} C_DIS
LIN {X 80.0642,Y 69.0327,Z 107,A 36.4193,B 24.927,C -1.9727,E1 25.1206,E2 409.1137} C_DIS
LIN {X 75.6701,Y 73.823,Z 107,A 40.1748,B 24.9257,C -1.9902,E1 25.1134,E2 405.3333} C_DIS
LIN {X 73.2475,Y 76.2249,Z 107,A 43.0052,B 24.9223,C -2.0355,E1 25.1075,E2 402.4074} C_DIS
LIN {X 68.6412,Y 80.3978,Z 107,A 44.8933,B 24.9265,C -1.98,E1 25.1038,E2 400.6579} C_DIS
LIN {X 65.053,Y 83.3301,Z 107,A 47.8164,B 24.9249,C -2.0017,E1 25.0973,E2 397.6946} C_DIS
LIN {X 62.353,Y 85.3669,Z 107,A 49.5345,B 24.9249,C -2.0002,E1 25.0935,E2 395.9862} C_DIS
LIN {X 59.9599,Y 87.0656,Z 107,A 52.0943,B 24.9217,C -2.0432,E1 25.0874,E2 393.3334} C_DIS
LIN {X 55.3502,Y 90.0668,Z 107,A 53.9698,B 24.9249,C -2.0019,E1 25.0832,E2 391.5616} C_DIS
LIN {X 50.8609,Y 92.676,Z 107,A 57.0002,B 24.9239,C -2.0147,E1 25.0758,E2 388.5099} C_DIS
LIN {X 47.7633,Y 94.3092,Z 107,A 58.9192,B 24.9236,C -2.0181,E1 25.071,E2 386.5882} C_DIS
LIN {X 45.0178,Y 95.6504,Z 107,A 61.2774,B 24.9213,C -2.0489,E1 25.0649,E2 384.1632} C_DIS
LIN {X 40.4822,Y 97.6574,Z 107,A 63.2702,B 24.9232,C -2.0232,E1 25.0599,E2 382.2358} C_DIS
LIN {X 35.452,Y 99.5931,Z 107,A 66.0273,B 24.9235,C -2.0194,E1 25.0528,E2 379.4938} C_DIS
LIN {X 31.6627,Y 100.8613,Z 107,A 68.2705,B 24.9232,C -2.0243,E1 25.0468,E2 377.2432} C_DIS
LIN {X 28.3547,Y 101.8413,Z 107,A 70.1045,B 24.9232,C -2.0241,E1 25.0419,E2 375.4127} C_DIS
LIN {X 25.0384,Y 102.7058,Z 107,A 71.854,B 24.9234,C -2.0209,E1 25.0372,E2 373.6733} C_DIS
LIN {X 22.0478,Y 103.3902,Z 107,A 73.7046,B 24.9228,C -2.0292,E1 25.0321,E2 371.8055} C_DIS
LIN {X 15.1985,Y 104.616,Z 107,A 77.3819,B 24.923,C -2.0268,E1 25.022,E2 368.1378} C_DIS
LIN {X 11.4098,Y 105.097,Z 107,A 79.9063,B 24.9216,C -2.0452,E1 25.0148,E2 365.5716} C_DIS
LIN {X 7.9008,Y 105.4194,Z 107,A 81.2104,B 24.9234,C -2.0213,E1 25.0114,E2 364.3248} C_DIS
LIN {X 2.2673,Y 105.6899,Z 107,A 84.4301,B 24.9229,C -2.0275,E1 25.0024,E2 361.0913} C_DIS
LIN {X -3.1363,Y 105.6673,Z 107,A 87.2597,B 24.9233,C -2.0229,E1 24.9945,E2 358.2725} C_DIS
LIN {X -8.3467,Y 105.3837,Z 107,A 90.1942,B 24.923,C -2.0259,E1 24.9863,E2 355.3299} C_DIS
LIN {X -11.4327,Y 105.0946,Z 107,A 92.6485,B 24.9208,C -2.0553,E1 24.9793,E2 352.8044} C_DIS
LIN {X -16.1798,Y 104.4682,Z 107,A 94.537,B 24.923,C -2.0259,E1 24.9742,E2 350.984} C_DIS
LIN {X -19.9687,Y 103.8106,Z 107,A 96.4471,B 24.9237,C -2.0176,E1 24.969,E2 349.0916} C_DIS
LIN {X -24.5483,Y 102.8253,Z 107,A 99.1127,B 24.9235,C -2.0202,E1 24.9618,E2 346.4165} C_DIS
LIN {X -27.6378,Y 102.037,Z 107,A 100.6972,B 24.924,C -2.013,E1 24.9575,E2 344.8469} C_DIS
LIN {X -33.6898,Y 100.2018,Z 107,A 104.531,B 24.9231,C -2.0245,E1 24.9472,E2 340.9789} C_DIS
LIN {X -39.5528,Y 98.0361,Z 107,A 107.7054,B 24.9241,C -2.0118,E1 24.939,E2 337.828} C_DIS
LIN {X -43.0106,Y 96.5696,Z 107,A 109.7723,B 24.9242,C -2.01,E1 24.9337,E2 335.7606} C_DIS
LIN {X -46.7405,Y 94.8197,Z 107,A 111.9987,B 24.9245,C -2.0063,E1 24.9281,E2 333.5374} C_DIS
LIN {X -50.1163,Y 93.0799,Z 107,A 114.0148,B 24.9249,C -2.0012,E1 24.9231,E2 331.5277} C_DIS
LIN {X -53.2,Y 91.3539,Z 107,A 116.784,B 24.9227,C -2.03,E1 24.9163,E2 328.6815} C_DIS
LIN {X -57.5056,Y 88.7059,Z 107,A 118.6024,B 24.9257,C -1.9901,E1 24.9122,E2 326.9525} C_DIS
LIN {X -59.8562,Y 87.1377,Z 107,A 121.1644,B 24.923,C -2.0258,E1 24.9061,E2 324.2967} C_DIS
LIN {X -64.2348,Y 83.9609,Z 107,A 123.1936,B 24.9261,C -1.9857,E1 24.9018,E2 322.3557} C_DIS
LIN {X -67.0261,Y 81.7512,Z 107,A 125.1834,B 24.9262,C -1.9837,E1 24.8974,E2 320.3632} C_DIS
LIN {X -70.747,Y 78.5517,Z 107,A 128.2615,B 24.9255,C -1.9932,E1 24.8909,E2 317.2503} C_DIS
LIN {X -73.3575,Y 76.1188,Z 107,A 129.728,B 24.9271,C -1.9713,E1 24.8881,E2 315.83} C_DIS
LIN {X -75.9328,Y 73.5505,Z 107,A 131.4216,B 24.9282,C -1.9563,E1 24.8848,E2 314.165} C_DIS
LIN {X -78.0352,Y 71.3158,Z 107,A 133.9896,B 24.9261,C -1.9855,E1 24.8798,E2 311.516} C_DIS
LIN {X -80.7834,Y 68.1885,Z 107,A 135.7022,B 24.928,C -1.9595,E1 24.8768,E2 309.8575} C_DIS
LIN {X -82.9335,Y 65.5548,Z 107,A 137.4947,B 24.9285,C -1.9528,E1 24.8736,E2 308.0725} C_DIS
LIN {X -84.9815,Y 62.8794,Z 107,A 139.3981,B 24.9287,C -1.9507,E1 24.8704,E2 306.1651} C_DIS
LIN {X -86.8872,Y 60.2165,Z 107,A 141.101,B 24.9292,C -1.9432,E1 24.8677,E2 304.4717} C_DIS
LIN {X -88.6065,Y 57.6601,Z 107,A 143.4432,B 24.9277,C -1.9632,E1 24.8641,E2 302.0701} C_DIS
LIN {X -90.81,Y 54.121,Z 107,A 145.0691,B 24.9299,C -1.9334,E1 24.8618,E2 300.5067} C_DIS
LIN {X -92.6469,Y 50.9145,Z 107,A 147.6062,B 24.9289,C -1.9471,E1 24.8583,E2 297.9237} C_DIS
LIN {X -94.375,Y 47.6344,Z 107,A 149.0204,B 24.9309,C -1.9194,E1 24.8566,E2 296.568} C_DIS
LIN {X -96.2057,Y 43.8183,Z 107,A 151.4663,B 24.931,C -1.918,E1 24.8537,E2 294.1121} C_DIS
LIN {X -97.6152,Y 40.5824,Z 107,A 153.9712,B 24.9299,C -1.9338,E1 24.8509,E2 291.5556} C_DIS
LIN {X -99.1348,Y 36.7146,Z 107,A 155.4634,B 24.9324,C -1.8991,E1 24.8495,E2 290.1378} C_DIS
LIN {X -100.7975,Y 31.865,Z 107,A 158.5344,B 24.9323,C -1.901,E1 24.8468,E2 287.0447} C_DIS
LIN {X -101.5886,Y 29.2463,Z 107,A 161.2342,B 24.9294,C -1.941,E1 24.8447,E2 284.2339} C_DIS
LIN {X -103.29,Y 22.5072,Z 107,A 163.666,B 24.9338,C -1.8799,E1 24.8432,E2 281.9335} C_DIS
LIN {X -103.9297,Y 19.3503,Z 107,A 165.4467,B 24.9341,C -1.8755,E1 24.8423,E2 280.1527} C_DIS
LIN {X -104.4422,Y 16.3479,Z 107,A 167.1633,B 24.9343,C -1.8726,E1 24.8415,E2 278.4328} C_DIS
LIN {X -104.9666,Y 12.5491,Z 107,A 169.2854,B 24.9346,C -1.8675,E1 24.8407,E2 276.3103} C_DIS
LIN {X -105.364,Y 8.5938,Z 107,A 172.4345,B 24.9325,C -1.8969,E1 24.84,E2 273.0721} C_DIS
LIN {X -105.681,Y 2.6901,Z 107,A 174.7428,B 24.9356,C -1.8537,E1 24.8398,E2 270.8531} C_DIS
LIN {X -105.7052,Y -1.439,Z 107,A 177.3415,B 24.9352,C -1.8596,E1 24.8398,E2 268.2246} C_DIS
LIN {X -105.5972,Y -4.9824,Z 107,A 178.8615,B 24.9366,C -1.8388,E1 24.84,E2 266.7451} C_DIS
LIN {X -105.3678,Y -8.546,Z 107,A -179.2454,B 24.9372,C -1.8311,E1 24.8404,E2 264.859} C_DIS
LIN {X -105.0683,Y -11.6807,Z 107,A -177.449,B 24.9373,C -1.8288,E1 24.841,E2 263.0572} C_DIS
LIN {X -104.6611,Y -14.881,Z 107,A -175.7772,B 24.9379,C -1.8205,E1 24.8416,E2 261.3953} C_DIS
LIN {X -104.1007,Y -18.3997,Z 107,A -173.8296,B 24.9383,C -1.815,E1 24.8425,E2 259.4491} C_DIS
LIN {X -103.4437,Y -21.797,Z 107,A -171.8471,B 24.9383,C -1.8131,E1 24.8436,E2 257.4597} C_DIS
LIN {X -102.6825,Y -25.1336,Z 107,A -170.0628,B 24.9389,C -1.8048,E1 24.8447,E2 255.6846} C_DIS
LIN {X -101.6197,Y -29.1366,Z 107,A -167.3131,B 24.9382,C -1.8164,E1 24.8468,E2 252.8912} C_DIS
LIN {X -100.5614,Y -32.6008,Z 107,A -165.8134,B 24.9397,C -1.7935,E1 24.8481,E2 251.4376} C_DIS
LIN {X -98.8642,Y -37.4334,Z 107,A -163.0429,B 24.9403,C -1.785,E1 24.8507,E2 248.6716} C_DIS
LIN {X -97.8582,Y -39.9899,Z 107,A -161.2679,B 24.9399,C -1.7912,E1 24.8526,E2 246.8719} C_DIS
LIN {X -96.0583,Y -44.1414,Z 107,A -158.9655,B 24.9407,C -1.7787,E1 24.8552,E2 244.5868} C_DIS
LIN {X -94.6544,Y -47.0739,Z 107,A -157.2802,B 24.9412,C -1.7709,E1 24.8572,E2 242.911} C_DIS
LIN {X -92.2676,Y -51.5954,Z 107,A -154.4007,B 24.9415,C -1.7673,E1 24.8611,E2 240.0248} C_DIS
LIN {X -90.0477,Y -55.3816,Z 107,A -151.819,B 24.9414,C -1.7685,E1 24.8648,E2 237.4269} C_DIS
LIN {X -87.58,Y -59.2042,Z 107,A -149.6795,B 24.9426,C -1.75,E1 24.8681,E2 235.3208} C_DIS
LIN {X -86.0659,Y -61.3845,Z 107,A -147.3247,B 24.9406,C -1.7808,E1 24.8721,E2 232.8812} C_DIS
LIN {X -82.9765,Y -65.5003,Z 107,A -145.4009,B 24.9432,C -1.7415,E1 24.8752,E2 231.042} C_DIS
LIN {X -80.4557,Y -68.5731,Z 107,A -142.8037,B 24.9424,C -1.7531,E1 24.8799,E2 228.4051} C_DIS
LIN {X -78.2051,Y -71.1307,Z 107,A -141.2214,B 24.9433,C -1.7389,E1 24.8828,E2 226.8495} C_DIS
LIN {X -75.9173,Y -73.5666,Z 107,A -139.3279,B 24.9433,C -1.7381,E1 24.8865,E2 224.9497} C_DIS
LIN {X -70.9333,Y -78.3849,Z 107,A -135.6911,B 24.9442,C -1.7258,E1 24.8939,E2 221.3275} C_DIS
LIN {X -68.8769,Y -80.1969,Z 107,A -133.937,B 24.9437,C -1.7331,E1 24.8976,E2 219.549} C_DIS
LIN {X -65.0683,Y -83.318,Z 107,A -131.5021,B 24.9446,C -1.7193,E1 24.9029,E2 217.138} C_DIS
LIN {X -58.7178,Y -87.9091,Z 107,A -127.2838,B 24.9451,C -1.7109,E1 24.9125,E2 212.925} C_DIS
LIN {X -56.3528,Y -89.4423,Z 107,A -125.4573,B 24.9446,C -1.7201,E1 24.9169,E2 211.0708} C_DIS
LIN {X -52.5989,Y -91.6993,Z 107,A -123.3022,B 24.9453,C -1.7082,E1 24.922,E2 208.9374} C_DIS
LIN {X -49.3196,Y -93.5039,Z 107,A -121.5977,B 24.9463,C -1.693,E1 24.9261,E2 207.2642} C_DIS
LIN {X -43.5747,Y -96.3155,Z 107,A -117.9717,B 24.9462,C -1.695,E1 24.9353,E2 203.6244} C_DIS
LIN {X -41.2259,Y -97.344,Z 107,A -116.252,B 24.9454,C -1.7063,E1 24.9398,E2 201.8736} C_DIS
LIN {X -37.317,Y -98.9083,Z 107,A -113.9799,B 24.9456,C -1.7038,E1 24.9457,E2 199.6028} C_DIS
LIN {X -32.8586,Y -100.478,Z 107,A -111.6522,B 24.9463,C -1.6925,E1 24.9518,E2 197.2975} C_DIS
LIN {X -29.5918,Y -101.4887,Z 107,A -109.7058,B 24.9462,C -1.6948,E1 24.957,E2 195.3423} C_DIS
LIN {X -25.825,Y -102.5121,Z 107,A -107.5838,B 24.9462,C -1.6938,E1 24.9627,E2 193.2196} C_DIS
LIN {X -18.4681,Y -104.0883,Z 107,A -103.5429,B 24.9464,C -1.6906,E1 24.9738,E2 189.1817} C_DIS
LIN {X -15.1028,Y -104.6296,Z 107,A -101.1522,B 24.9451,C -1.7119,E1 24.9805,E2 186.7384} C_DIS
LIN {X -11.0338,Y -105.1363,Z 107,A -99.934,B 24.9476,C -1.6714,E1 24.9837,E2 185.6154} C_DIS
LIN {X -7.6913,Y -105.4337,Z 107,A -97.526,B 24.9462,C -1.6949,E1 24.9905,E2 183.1508} C_DIS
LIN {X 0.418,Y -105.7132,Z 107,A -93.6164,B 24.9474,C -1.6758,E1 25.0013,E2 179.2859} C_DIS
LIN {X 0.418,Y -105.7132,Z 107,A -93.6164,B 24.9474,C -1.6758,E1 25.0013,E2 179.2859} C_DIS
Enddeposition()
LIN {X 0.7311,Y -104.7335,Z 107,A -94.3847,B 24.9486,C -1.656,E1 24.999,E2 180.1011} C_DIS
Startdeposition()
$VEL.CP = VEL_PRINT
LIN {X -3.1167,Y -104.7024,Z 107,A -96.0909,B 24.9477,C -1.671,E1 24.9944,E2 181.7719} C_DIS
LIN {X -5.5843,Y -104.5999,Z 107,A -98.0712,B 24.9492,C -1.6464,E1 24.9887,E2 183.8109} C_DIS
LIN {X -9.6476,Y -104.3035,Z 107,A -99.6622,B 24.9477,C -1.6712,E1 24.9844,E2 185.344} C_DIS
LIN {X -13.9132,Y -103.8216,Z 107,A -101.9574,B 24.9475,C -1.6736,E1 24.9781,E2 187.635} C_DIS
LIN {X -16.8036,Y -103.3932,Z 107,A -103.7811,B 24.948,C -1.6653,E1 24.973,E2 189.48} C_DIS
LIN {X -22.7008,Y -102.26,Z 107,A -107.0267,B 24.9478,C -1.6682,E1 24.9641,E2 192.7226} C_DIS
LIN {X -26.3904,Y -101.3703,Z 107,A -108.9795,B 24.9475,C -1.6741,E1 24.9588,E2 194.664} C_DIS
LIN {X -29.6312,Y -100.4705,Z 107,A -110.8329,B 24.9475,C -1.6748,E1 24.9539,E2 196.5188} C_DIS
LIN {X -32.9932,Y -99.4183,Z 107,A -112.6483,B 24.9471,C -1.6805,E1 24.9491,E2 198.3238} C_DIS
LIN {X -36.0064,Y -98.3659,Z 107,A -114.589,B 24.9474,C -1.6746,E1 24.9439,E2 200.2824} C_DIS
LIN {X -39.1035,Y -97.1771,Z 107,A -116.4084,B 24.9474,C -1.6762,E1 24.9392,E2 202.102} C_DIS
LIN {X -42.4631,Y -95.7579,Z 107,A -118.445,B 24.9474,C -1.6768,E1 24.9339,E2 204.142} C_DIS
LIN {X -47.5949,Y -93.3114,Z 107,A -121.447,B 24.9468,C -1.6846,E1 24.9264,E2 207.1333} C_DIS
LIN {X -50.0553,Y -92.0151,Z 107,A -122.9158,B 24.9466,C -1.6886,E1 24.9228,E2 208.5967} C_DIS
LIN {X -52.8342,Y -90.4496,Z 107,A -124.8969,B 24.947,C -1.6822,E1 24.918,E2 210.5989} C_DIS
LIN {X -56.0069,Y -88.5205,Z 107,A -126.6942,B 24.9462,C -1.694,E1 24.9138,E2 212.3739} C_DIS
LIN {X -58.2336,Y -87.0718,Z 107,A -128.124,B 24.946,C -1.6971,E1 24.9104,E2 213.8008} C_DIS
LIN {X -62.1543,Y -84.3164,Z 107,A -130.9604,B 24.9462,C -1.6936,E1 24.904,E2 216.6554} C_DIS
LIN {X -65.5713,Y -81.6881,Z 107,A -133.4621,B 24.9463,C -1.6926,E1 24.8984,E2 219.1687} C_DIS
LIN {X -68.8314,Y -78.9591,Z 107,A -135.5704,B 24.9455,C -1.7051,E1 24.894,E2 221.2556} C_DIS
LIN {X -70.855,Y -77.1483,Z 107,A -138.1736,B 24.9479,C -1.6675,E1 24.8885,E2 223.9588} C_DIS
LIN {X -75.2146,Y -72.905,Z 107,A -140.1369,B 24.9443,C -1.724,E1 24.8849,E2 225.7958} C_DIS
LIN {X -78.921,Y -68.875,Z 107,A -143.4148,B 24.9445,C -1.7204,E1 24.8787,E2 229.0969} C_DIS
LIN {X -81.1655,Y -66.2161,Z 107,A -145.3718,B 24.9444,C -1.7229,E1 24.8752,E2 231.057} C_DIS
LIN {X -83.1078,Y -63.7608,Z 107,A -147.5096,B 24.9451,C -1.7117,E1 24.8715,E2 233.2317} C_DIS
LIN {X -85.177,Y -60.9688,Z 107,A -148.9504,B 24.9437,C -1.7329,E1 24.8692,E2 234.6288} C_DIS
LIN {X -87.1126,Y -58.1727,Z 107,A -150.7238,B 24.9432,C -1.7408,E1 24.8664,E2 236.3923} C_DIS
LIN {X -88.7779,Y -55.5949,Z 107,A -152.5244,B 24.9432,C -1.7408,E1 24.8637,E2 238.202} C_DIS
LIN {X -90.6107,Y -52.5563,Z 107,A -154.8423,B 24.9437,C -1.7325,E1 24.8603,E2 240.5518} C_DIS
LIN {X -93.092,Y -48.0242,Z 107,A -157.443,B 24.9427,C -1.7483,E1 24.857,E2 243.1285} C_DIS
LIN {X -94.9227,Y -44.2943,Z 107,A -159.565,B 24.9419,C -1.7601,E1 24.8544,E2 245.2339} C_DIS
LIN {X -95.9422,Y -42.0407,Z 107,A -161.1196,B 24.9422,C -1.7568,E1 24.8526,E2 246.805} C_DIS
LIN {X -97.4424,Y -38.4356,Z 107,A -163.0713,B 24.9413,C -1.7695,E1 24.8506,E2 248.7371} C_DIS
LIN {X -99.5338,Y -32.6418,Z 107,A -166.2962,B 24.9403,C -1.7847,E1 24.8476,E2 251.9442} C_DIS
LIN {X -100.9104,Y -28.0999,Z 107,A -169.2043,B 24.9405,C -1.7814,E1 24.8453,E2 254.8769} C_DIS
LIN {X -101.7771,Y -24.7733,Z 107,A -170.9763,B 24.9399,C -1.7911,E1 24.8441,E2 256.6362} C_DIS
LIN {X -102.5769,Y -21.2202,Z 107,A -173.0167,B 24.9396,C -1.7956,E1 24.8429,E2 258.6779} C_DIS
LIN {X -103.2686,Y -17.549,Z 107,A -175.1226,B 24.9393,C -1.7998,E1 24.8418,E2 260.7863} C_DIS
LIN {X -103.8498,Y -13.6952,Z 107,A -177.1409,B 24.9386,C -1.8105,E1 24.841,E2 262.791} C_DIS
LIN {X -104.1579,Y -11.1111,Z 107,A -178.6519,B 24.9385,C -1.812,E1 24.8406,E2 264.3076} C_DIS
LIN {X -104.4727,Y -7.6199,Z 107,A 179.3496,B 24.9382,C -1.8152,E1 24.8401,E2 266.3103} C_DIS
LIN {X -104.6476,Y -4.6033,Z 107,A 177.5568,B 24.9382,C -1.8156,E1 24.8399,E2 268.1129} C_DIS
LIN {X -104.747,Y -0.5828,Z 107,A 175.593,B 24.9372,C -1.831,E1 24.8398,E2 270.0518} C_DIS
LIN {X -104.7218,Y 2.4283,Z 107,A 173.9589,B 24.9368,C -1.8368,E1 24.8398,E2 271.682} C_DIS
LIN {X -104.4519,Y 7.8935,Z 107,A 170.7697,B 24.9366,C -1.8396,E1 24.8404,E2 274.8838} C_DIS
LIN {X -104.0892,Y 11.7438,Z 107,A 168.6933,B 24.936,C -1.8478,E1 24.841,E2 276.953} C_DIS
LIN {X -103.6535,Y 15.1122,Z 107,A 166.7658,B 24.9358,C -1.8513,E1 24.8417,E2 278.8836} C_DIS
LIN {X -103.0487,Y 18.797,Z 107,A 164.8001,B 24.9351,C -1.8606,E1 24.8426,E2 280.8389} C_DIS
LIN {X -102.4741,Y 21.7193,Z 107,A 162.999,B 24.9351,C -1.8597,E1 24.8436,E2 282.6526} C_DIS
LIN {X -100.9423,Y 27.9875,Z 107,A 159.4978,B 24.9343,C -1.8719,E1 24.8461,E2 286.1451} C_DIS
LIN {X -100.0956,Y 30.8737,Z 107,A 157.1471,B 24.9357,C -1.8525,E1 24.8481,E2 288.5556} C_DIS
LIN {X -98.5523,Y 35.4953,Z 107,A 155.2085,B 24.9333,C -1.8862,E1 24.8498,E2 290.425} C_DIS
LIN {X -96.8795,Y 39.8345,Z 107,A 152.7434,B 24.9326,C -1.8968,E1 24.8523,E2 292.8786} C_DIS
LIN {X -95.6095,Y 42.7924,Z 107,A 150.9443,B 24.9323,C -1.9008,E1 24.8543,E2 294.6781} C_DIS
LIN {X -94.0882,Y 46.0433,Z 107,A 148.3261,B 24.9335,C -1.8836,E1 24.8576,E2 297.3513} C_DIS
LIN {X -92.2088,Y 49.6981,Z 107,A 146.5946,B 24.9317,C -1.9084,E1 24.8598,E2 299.033} C_DIS
LIN {X -90.1595,Y 53.325,Z 107,A 143.795,B 24.9326,C -1.8967,E1 24.8638,E2 301.8751} C_DIS
LIN {X -88.0161,Y 56.7936,Z 107,A 142.0518,B 24.9309,C -1.9201,E1 24.8663,E2 303.5712} C_DIS
LIN {X -85.9183,Y 59.9197,Z 107,A 140.0562,B 24.9303,C -1.9281,E1 24.8695,E2 305.5577} C_DIS
LIN {X -83.7453,Y 62.9208,Z 107,A 138.0887,B 24.9298,C -1.9357,E1 24.8727,E2 307.5166} C_DIS
LIN {X -81.5261,Y 65.7712,Z 107,A 136.0926,B 24.9294,C -1.9402,E1 24.8762,E2 309.5113} C_DIS
LIN {X -79.6273,Y 68.0574,Z 107,A 134.1646,B 24.9299,C -1.9337,E1 24.8797,E2 311.4637} C_DIS
LIN {X -76.499,Y 71.5561,Z 107,A 131.7843,B 24.9289,C -1.9468,E1 24.8841,E2 313.8233} C_DIS
LIN {X -73.8876,Y 74.25,Z 107,A 129.7052,B 24.9286,C -1.9508,E1 24.8882,E2 315.9017} C_DIS
LIN {X -71.9746,Y 76.1054,Z 107,A 128.2087,B 24.9285,C -1.9529,E1 24.8912,E2 317.3994} C_DIS
LIN {X -68.4554,Y 79.2875,Z 107,A 125.5855,B 24.9281,C -1.9578,E1 24.8967,E2 320.0212} C_DIS
LIN {X -65.4412,Y 81.7932,Z 107,A 123.5021,B 24.9276,C -1.9647,E1 24.9012,E2 322.0961} C_DIS
LIN {X -62.9077,Y 83.7551,Z 107,A 121.2606,B 24.9286,C -1.9508,E1 24.9063,E2 324.3788} C_DIS
LIN {X -59.8573,Y 85.9616,Z 107,A 119.6946,B 24.927,C -1.9728,E1 24.9098,E2 325.8979} C_DIS
LIN {X -57.3773,Y 87.637,Z 107,A 118.1031,B 24.9267,C -1.9776,E1 24.9134,E2 327.4832} C_DIS
LIN {X -54.4863,Y 89.4625,Z 107,A 115.7611,B 24.9277,C -1.964,E1 24.9191,E2 329.8649} C_DIS
LIN {X -51.4953,Y 91.2182,Z 107,A 114.2343,B 24.9264,C -1.9808,E1 24.9227,E2 331.3562} C_DIS
LIN {X -48.5424,Y 92.8225,Z 107,A 112.5819,B 24.9257,C -1.9907,E1 24.9267,E2 332.9897} C_DIS
LIN {X -44.9846,Y 94.5984,Z 107,A 110.2567,B 24.9259,C -1.9886,E1 24.9326,E2 335.3258} C_DIS
LIN {X -41.7131,Y 96.085,Z 107,A 108.2525,B 24.9257,C -1.9902,E1 24.9377,E2 337.3312} C_DIS
LIN {X -38.7073,Y 97.3357,Z 107,A 105.7665,B 24.9275,C -1.9667,E1 24.9443,E2 339.8783} C_DIS
LIN {X -34.4062,Y 98.9373,Z 107,A 103.8081,B 24.9257,C -1.9902,E1 24.9493,E2 341.7849} C_DIS
LIN {X -27.9117,Y 100.9634,Z 107,A 100.16,B 24.9252,C -1.997,E1 24.9591,E2 345.4229} C_DIS
LIN {X -24.6343,Y 101.811,Z 107,A 98.1554,B 24.9255,C -1.9931,E1 24.9645,E2 347.4395} C_DIS
LIN {X -20.017,Y 102.8186,Z 107,A 95.8478,B 24.9246,C -2.0057,E1 24.9708,E2 349.72} C_DIS
LIN {X -16.8131,Y 103.3916,Z 107,A 94.1981,B 24.9241,C -2.0119,E1 24.9753,E2 351.3565} C_DIS
LIN {X -13.011,Y 103.9385,Z 107,A 92.0144,B 24.9242,C -2.0101,E1 24.9813,E2 353.5462} C_DIS
LIN {X -10.2113,Y 104.2514,Z 107,A 90.2364,B 24.9249,C -2.002,E1 24.9863,E2 355.3445} C_DIS
LIN {X -5.4591,Y 104.6068,Z 107,A 87.547,B 24.925,C -1.9999,E1 24.9938,E2 358.0398} C_DIS
LIN {X -0.9727,Y 104.7447,Z 107,A 85.3312,B 24.9243,C -2.0097,E1 25,E2 360.2326} C_DIS
LIN {X 2.2153,Y 104.7257,Z 107,A 83.7003,B 24.9239,C -2.0143,E1 25.0045,E2 361.8524} C_DIS
LIN {X 6.5248,Y 104.5463,Z 107,A 81.2952,B 24.9241,C -2.0126,E1 25.0112,E2 364.2607} C_DIS
LIN {X 10.1853,Y 104.2539,Z 107,A 79.2287,B 24.9242,C -2.0102,E1 25.017,E2 366.3319} C_DIS
LIN {X 13.2809,Y 103.9035,Z 107,A 77.5085,B 24.9243,C -2.0092,E1 25.0217,E2 368.053} C_DIS
LIN {X 15.6589,Y 103.5723,Z 107,A 75.7697,B 24.9256,C -1.9924,E1 25.0266,E2 369.8299} C_DIS
LIN {X 18.9763,Y 103.0164,Z 107,A 74.2923,B 24.9246,C -2.0057,E1 25.0306,E2 371.2743} C_DIS
LIN {X 22.1751,Y 102.3747,Z 107,A 72.5781,B 24.9244,C -2.0076,E1 25.0353,E2 372.9817} C_DIS
LIN {X 25.4407,Y 101.6138,Z 107,A 70.6588,B 24.9248,C -2.0032,E1 25.0405,E2 374.9086} C_DIS
LIN {X 28.886,Y 100.6877,Z 107,A 68.6955,B 24.9248,C -2.0015,E1 25.0458,E2 376.873} C_DIS
LIN {X 32.9701,Y 99.4258,Z 107,A 66.4313,B 24.9248,C -2.0025,E1 25.0518,E2 379.1305} C_DIS
LIN {X 36.4494,Y 98.2043,Z 107,A 64.521,B 24.9246,C -2.0049,E1 25.0568,E2 381.0313} C_DIS
LIN {X 39.319,Y 97.0893,Z 107,A 62.7523,B 24.925,C -1.9999,E1 25.0614,E2 382.8079} C_DIS
LIN {X 44.1757,Y 94.9779,Z 107,A 59.8902,B 24.9252,C -1.998,E1 25.0687,E2 385.6675} C_DIS
LIN {X 47.2506,Y 93.4874,Z 107,A 58.0181,B 24.9253,C -1.9955,E1 25.0734,E2 387.5404} C_DIS
LIN {X 50.2892,Y 91.8882,Z 107,A 55.7807,B 24.9266,C -1.9786,E1 25.079,E2 389.8113} C_DIS
LIN {X 54.2633,Y 89.5981,Z 107,A 53.6144,B 24.9259,C -1.9886,E1 25.0841,E2 391.9473} C_DIS
LIN {X 59.3843,Y 86.2904,Z 107,A 50.2263,B 24.9264,C -1.9811,E1 25.092,E2 395.342} C_DIS
LIN {X 62.4636,Y 84.0887,Z 107,A 48.381,B 24.926,C -1.9866,E1 25.0961,E2 397.1678} C_DIS
LIN {X 65.8863,Y 81.4327,Z 107,A 45.924,B 24.9266,C -1.9787,E1 25.1016,E2 399.6343} C_DIS
LIN {X 68.1081,Y 79.5842,Z 107,A 43.9578,B 24.928,C -1.96,E1 25.1058,E2 401.637} C_DIS
LIN {X 73.2022,Y 74.927,Z 107,A 40.5058,B 24.9276,C -1.9653,E1 25.1128,E2 405.0623} C_DIS
LIN {X 77.1622,Y 70.8398,Z 107,A 37.413,B 24.928,C -1.9593,E1 25.1188,E2 408.1559} C_DIS
LIN {X 79.9344,Y 67.697,Z 107,A 34.5634,B 24.9301,C -1.9313,E1 25.124,E2 411.0589} C_DIS
LIN {X 82.576,Y 64.4508,Z 107,A 32.8387,B 24.9288,C -1.9488,E1 25.1269,E2 412.7341} C_DIS
LIN {X 84.4378,Y 61.9884,Z 107,A 31.2445,B 24.9288,C -1.9485,E1 25.1296,E2 414.3212} C_DIS
LIN {X 88.5122,Y 56.0202,Z 107,A 27.1765,B 24.9299,C -1.9336,E1 25.1359,E2 418.4044} C_DIS
LIN {X 91.6205,Y 50.7748,Z 107,A 23.9141,B 24.9303,C -1.9276,E1 25.1405,E2 421.664} C_DIS
LIN {X 93.3931,Y 47.435,Z 107,A 22.1498,B 24.9298,C -1.9345,E1 25.1428,E2 423.4027} C_DIS
LIN {X 96.4537,Y 40.8534,Z 107,A 17.9702,B 24.9313,C -1.9144,E1 25.1477,E2 427.6071} C_DIS
LIN {X 98.8257,Y 34.7242,Z 107,A 14.4337,B 24.9319,C -1.9062,E1 25.1512,E2 431.1432} C_DIS
LIN {X 99.8441,Y 31.6829,Z 107,A 12.5696,B 24.9326,C -1.8963,E1 25.1528,E2 433.0201} C_DIS
LIN {X 100.851,Y 28.3096,Z 107,A 10.8825,B 24.9323,C -1.9005,E1 25.1541,E2 434.6878} C_DIS
LIN {X 101.5919,Y 25.5285,Z 107,A 9.16,B 24.9331,C -1.8894,E1 25.1553,E2 436.4265} C_DIS
LIN {X 102.4843,Y 21.6714,Z 107,A 6.8624,B 24.9339,C -1.8771,E1 25.1567,E2 438.7397} C_DIS
LIN {X 103.4246,Y 16.614,Z 107,A 4.1514,B 24.9343,C -1.8726,E1 25.158,E2 441.4455} C_DIS
LIN {X 103.8638,Y 13.5873,Z 107,A 2.5327,B 24.9345,C -1.8696,E1 25.1586,E2 443.0618} C_DIS
LIN {X 104.158,Y 11.111,Z 107,A 0.7634,B 24.936,C -1.8482,E1 25.1591,E2 444.871} C_DIS
LIN {X 104.4747,Y 7.5894,Z 107,A -0.5562,B 24.9346,C -1.8678,E1 25.1594,E2 446.1366} C_DIS
LIN {X 104.7463,Y 0.7161,Z 107,A -5.2011,B 24.938,C -1.8186,E1 25.1598,E2 450.8698} C_DIS
LIN {X 104.6721,Y -4.0317,Z 107,A -7.4505,B 24.9376,C -1.8247,E1 25.1596,E2 453.0916} C_DIS
LIN {X 104.4898,Y -7.3668,Z 107,A -8.8662,B 24.9368,C -1.8361,E1 25.1593,E2 454.4719} C_DIS
LIN {X 104.1153,Y -11.5183,Z 107,A -11.494,B 24.9383,C -1.814,E1 25.1585,E2 457.1362} C_DIS
LIN {X 103.4515,Y -16.4398,Z 107,A -13.7642,B 24.9376,C -1.824,E1 25.1576,E2 459.3694} C_DIS
LIN {X 102.8355,Y -19.9293,Z 107,A -15.6373,B 24.9379,C -1.8206,E1 25.1567,E2 461.2397} C_DIS
LIN {X 102.2392,Y -22.7962,Z 107,A -17.2759,B 24.9383,C -1.8138,E1 25.1557,E2 462.8847} C_DIS
LIN {X 101.527,Y -25.7808,Z 107,A -19.2638,B 24.9396,C -1.7954,E1 25.1544,E2 464.9045} C_DIS
LIN {X 100.2716,Y -30.3016,Z 107,A -21.4194,B 24.939,C -1.8046,E1 25.1527,E2 467.0262} C_DIS
LIN {X 99.3055,Y -33.3275,Z 107,A -23.34,B 24.9398,C -1.7914,E1 25.151,E2 468.967} C_DIS
LIN {X 96.6653,Y -40.3513,Z 107,A -27.3661,B 24.9405,C -1.782,E1 25.147,E2 472.9929} C_DIS
LIN {X 93.102,Y -48.0047,Z 107,A -31.908,B 24.9412,C -1.7712,E1 25.1416,E2 477.5357} C_DIS
LIN {X 91.4823,Y -51.0224,Z 107,A -33.7213,B 24.9414,C -1.7683,E1 25.1391,E2 479.3466} C_DIS
LIN {X 90.0662,Y -53.4828,Z 107,A -35.4181,B 24.9421,C -1.7577,E1 25.1367,E2 481.0596} C_DIS
LIN {X 87.8384,Y -57.0704,Z 107,A -37.5951,B 24.9421,C -1.7566,E1 25.1335,E2 483.2281} C_DIS
LIN {X 86.1766,Y -59.5481,Z 107,A -39.5039,B 24.9432,C -1.7405,E1 25.1304,E2 485.1655} C_DIS
LIN {X 81.9056,Y -65.299,Z 107,A -43.1947,B 24.9432,C -1.7394,E1 25.1242,E2 488.8415} C_DIS
LIN {X 79.8546,Y -67.7906,Z 107,A -45.5623,B 24.9452,C -1.7098,E1 25.1198,E2 491.2681} C_DIS
LIN {X 76.9736,Y -71.0454,Z 107,A -47.1078,B 24.9434,C -1.7382,E1 25.1171,E2 492.7396} C_DIS
LIN {X 73.038,Y -75.0864,Z 107,A -50.156,B 24.9438,C -1.7321,E1 25.1111,E2 495.7893} C_DIS
LIN {X 68.8206,Y -78.9685,Z 107,A -53.2244,B 24.9441,C -1.7275,E1 25.1048,E2 498.8561} C_DIS
LIN {X 65.5636,Y -81.6943,Z 107,A -55.8218,B 24.9451,C -1.7109,E1 25.0991,E2 501.4828} C_DIS
LIN {X 63.3184,Y -83.4465,Z 107,A -57.8254,B 24.9465,C -1.6892,E1 25.0946,E2 503.5302} C_DIS
LIN {X 60.3111,Y -85.6455,Z 107,A -59.52,B 24.9459,C -1.6991,E1 25.0908,E2 505.1958} C_DIS
LIN {X 56.7355,Y -88.0534,Z 107,A -61.6396,B 24.9456,C -1.7042,E1 25.0859,E2 507.2961} C_DIS
LIN {X 54.3136,Y -89.5675,Z 107,A -63.1693,B 24.9456,C -1.7026,E1 25.0823,E2 508.8248} C_DIS
LIN {X 51.9816,Y -90.941,Z 107,A -65.352,B 24.9477,C -1.6713,E1 25.0768,E2 511.075} C_DIS
LIN {X 48.2303,Y -92.9867,Z 107,A -67.1279,B 24.9465,C -1.69,E1 25.0725,E2 512.8016} C_DIS
LIN {X 45.1739,Y -94.5074,Z 107,A -68.983,B 24.9466,C -1.6875,E1 25.0679,E2 514.6577} C_DIS
LIN {X 37.7169,Y -97.7247,Z 107,A -73.2327,B 24.9466,C -1.6888,E1 25.057,E2 518.8945} C_DIS
LIN {X 30.8626,Y -100.0991,Z 107,A -77.188,B 24.9468,C -1.6842,E1 25.0465,E2 522.8528} C_DIS
LIN {X 27.9014,Y -100.9662,Z 107,A -79.0707,B 24.9475,C -1.6745,E1 25.0414,E2 524.7554} C_DIS
LIN {X 24.705,Y -101.7938,Z 107,A -80.7735,B 24.9473,C -1.6768,E1 25.0368,E2 526.4502} C_DIS
LIN {X 20.9398,Y -102.6345,Z 107,A -82.8241,B 24.9473,C -1.6773,E1 25.0312,E2 528.4969} C_DIS
LIN {X 17.9597,Y -103.1993,Z 107,A -84.5631,B 24.9476,C -1.6727,E1 25.0264,E2 530.2448} C_DIS
LIN {X 15.5411,Y -103.5905,Z 107,A -86.0698,B 24.948,C -1.6652,E1 25.0222,E2 531.768} C_DIS
LIN {X 10.4932,Y -104.2226,Z 107,A -88.7445,B 24.9479,C -1.6678,E1 25.0148,E2 534.4346} C_DIS
LIN {X 7.0659,Y -104.5101,Z 107,A -90.5211,B 24.9477,C -1.671,E1 25.0099,E2 536.2026} C_DIS
LIN {X 1.466,Y -104.7395,Z 107,A -94.3476,B 24.9496,C -1.6403,E1 24.999,E2 540.1011} C_DIS
LIN {X 1.466,Y -104.7395,Z 107,A -94.3476,B 24.9496,C -1.6403,E1 24.999,E2 540.1011} C_DIS
Enddeposition()
LIN {X 0.7183,Y -103.7767,Z 107,A -93.2942,B 24.9449,C -1.7144,E1 25.0025,E2 538.8722} C_DIS
Startdeposition()
$VEL.CP = VEL_PRINT
LIN {X 4.3963,Y -103.6905,Z 107,A -91.1892,B 24.9447,C -1.7179,E1 25.0084,E2 536.7593} C_DIS
LIN {X 7.9356,Y -103.4804,Z 107,A -89.1906,B 24.9445,C -1.7204,E1 25.0139,E2 534.7556} C_DIS
LIN {X 11.6919,Y -103.1237,Z 107,A -86.9446,B 24.944,C -1.7281,E1 25.0202,E2 532.493} C_DIS
LIN {X 15.2862,Y -102.6534,Z 107,A -85.2747,B 24.9448,C -1.7162,E1 25.0248,E2 530.8527} C_DIS
LIN {X 18.3871,Y -102.1419,Z 107,A -83.3485,B 24.9442,C -1.7253,E1 25.0301,E2 528.9072} C_DIS
LIN {X 21.3835,Y -101.5581,Z 107,A -81.6077,B 24.944,C -1.7289,E1 25.0349,E2 527.1598} C_DIS
LIN {X 24.67,Y -100.809,Z 107,A -79.8741,B 24.9442,C -1.7256,E1 25.0396,E2 525.4365} C_DIS
LIN {X 27.6348,Y -100.0386,Z 107,A -78.2903,B 24.9444,C -1.7231,E1 25.0438,E2 523.8612} C_DIS
LIN {X 30.8963,Y -99.0782,Z 107,A -76.0947,B 24.9434,C -1.7382,E1 25.0498,E2 521.6338} C_DIS
LIN {X 36.6883,Y -97.0825,Z 107,A -73.037,B 24.9439,C -1.7294,E1 25.0578,E2 518.6031} C_DIS
LIN {X 39.6472,Y -95.9138,Z 107,A -71.0725,B 24.9432,C -1.7404,E1 25.0629,E2 516.6171} C_DIS
LIN {X 45.1601,Y -93.4434,Z 107,A -67.929,B 24.9434,C -1.7377,E1 25.0708,E2 513.4879} C_DIS
LIN {X 48.3217,Y -91.848,Z 107,A -65.7955,B 24.9427,C -1.7483,E1 25.0762,E2 511.3352} C_DIS
LIN {X 51.0745,Y -90.3479,Z 107,A -64.0979,B 24.9427,C -1.75,E1 25.0803,E2 509.6385} C_DIS
LIN {X 54.4047,Y -88.3828,Z 107,A -62.1741,B 24.9429,C -1.7453,E1 25.0849,E2 507.7318} C_DIS
LIN {X 57.6965,Y -86.27,Z 107,A -60.0387,B 24.9427,C -1.7485,E1 25.0899,E2 505.5958} C_DIS
LIN {X 60.2691,Y -84.4907,Z 107,A -58.1922,B 24.9421,C -1.7571,E1 25.0941,E2 503.7355} C_DIS
LIN {X 63.0653,Y -82.4254,Z 107,A -56.2043,B 24.9417,C -1.764,E1 25.0986,E2 501.7385} C_DIS
LIN {X 66.1604,Y -79.9619,Z 107,A -54.088,B 24.9415,C -1.766,E1 25.1032,E2 499.6254} C_DIS
LIN {X 69.3869,Y -77.1787,Z 107,A -51.5628,B 24.9407,C -1.7787,E1 25.1085,E2 497.0804} C_DIS
LIN {X 72.5299,Y -74.2347,Z 107,A -49.3038,B 24.9407,C -1.7794,E1 25.113,E2 494.8289} C_DIS
LIN {X 74.9328,Y -71.8068,Z 107,A -47.1095,B 24.9395,C -1.797,E1 25.1173,E2 492.6024} C_DIS
LIN {X 77.2016,Y -69.3613,Z 107,A -45.5961,B 24.9401,C -1.7879,E1 25.1201,E2 491.1172} C_DIS
LIN {X 79.7275,Y -66.4424,Z 107,A -43.59,B 24.9401,C -1.7883,E1 25.1237,E2 489.1196} C_DIS
LIN {X 82.0189,Y -63.5927,Z 107,A -41.6028,B 24.9398,C -1.7923,E1 25.1272,E2 487.132} C_DIS
LIN {X 84.3433,Y -60.4758,Z 107,A -39.4375,B 24.9393,C -1.799,E1 25.1308,E2 484.9613} C_DIS
LIN {X 86.2547,Y -57.7191,Z 107,A -37.4754,B 24.9387,C -1.8088,E1 25.1339,E2 482.9858} C_DIS
LIN {X 88.4075,Y -54.3641,Z 107,A -35.559,B 24.9391,C -1.8031,E1 25.1367,E2 481.0925} C_DIS
LIN {X 89.7579,Y -52.1036,Z 107,A -33.9197,B 24.9382,C -1.8152,E1 25.139,E2 479.4332} C_DIS
LIN {X 91.4874,Y -49.0042,Z 107,A -32.1271,B 24.9383,C -1.8139,E1 25.1414,E2 477.653} C_DIS
LIN {X 92.4578,Y -47.1446,Z 107,A -30.5084,B 24.9368,C -1.8369,E1 25.1435,E2 475.9886} C_DIS
LIN {X 94.7418,Y -42.369,Z 107,A -28.0465,B 24.9375,C -1.8262,E1 25.1464,E2 473.5653} C_DIS
LIN {X 95.8859,Y -39.7159,Z 107,A -26.4224,B 24.9371,C -1.8323,E1 25.1481,E2 471.9358} C_DIS
LIN {X 97.1117,Y -36.6114,Z 107,A -24.5062,B 24.9365,C -1.8412,E1 25.1501,E2 470.0094} C_DIS
LIN {X 99.1977,Y -30.5109,Z 107,A -21.0845,B 24.9361,C -1.8465,E1 25.1531,E2 466.5945} C_DIS
LIN {X 100.2752,Y -26.7587,Z 107,A -18.9216,B 24.9356,C -1.8536,E1 25.1547,E2 464.427} C_DIS
LIN {X 100.9108,Y -24.2525,Z 107,A -17.3472,B 24.9348,C -1.8644,E1 25.1558,E2 462.8363} C_DIS
LIN {X 101.7868,Y -20.27,Z 107,A -15.3226,B 24.935,C -1.862,E1 25.1569,E2 460.8292} C_DIS
LIN {X 102.3532,Y -17.1721,Z 107,A -13.4393,B 24.9342,C -1.8738,E1 25.1578,E2 458.9291} C_DIS
LIN {X 102.8086,Y -14.1991,Z 107,A -11.8943,B 24.9342,C -1.8742,E1 25.1584,E2 457.3921} C_DIS
LIN {X 103.108,Y -11.8255,Z 107,A -10.5554,B 24.9338,C -1.8793,E1 25.1589,E2 456.0493} C_DIS
LIN {X 103.4424,Y -8.4104,Z 107,A -8.647,B 24.9333,C -1.886,E1 25.1594,E2 454.1363} C_DIS
LIN {X 103.6631,Y -5.0357,Z 107,A -6.6159,B 24.9324,C -1.899,E1 25.1597,E2 452.0866} C_DIS
LIN {X 103.7837,Y -0.2638,Z 107,A -4.2055,B 24.9324,C -1.898,E1 25.1597,E2 449.693} C_DIS
LIN {X 103.727,Y 3.4391,Z 107,A -1.7801,B 24.9308,C -1.9208,E1 25.1596,E2 447.2282} C_DIS
LIN {X 103.4591,Y 8.2018,Z 107,A 0.4659,B 24.9314,C -1.9128,E1 25.1592,E2 445.0145} C_DIS
LIN {X 103.2185,Y 10.816,Z 107,A 1.9428,B 24.931,C -1.9186,E1 25.1588,E2 443.5325} C_DIS
LIN {X 102.7817,Y 14.3883,Z 107,A 3.9452,B 24.9305,C -1.9256,E1 25.158,E2 441.5255} C_DIS
LIN {X 102.1626,Y 18.2721,Z 107,A 6.0007,B 24.9303,C -1.9275,E1 25.1571,E2 439.4775} C_DIS
LIN {X 101.664,Y 20.8683,Z 107,A 7.5476,B 24.9297,C -1.9358,E1 25.1562,E2 437.9202} C_DIS
LIN {X 101.0019,Y 23.8735,Z 107,A 9.2998,B 24.9292,C -1.9433,E1 25.1551,E2 436.1604} C_DIS
LIN {X 100.1291,Y 27.2998,Z 107,A 11.0536,B 24.9294,C -1.9409,E1 25.1539,E2 434.4222} C_DIS
LIN {X 99.1695,Y 30.602,Z 107,A 13.0438,B 24.9287,C -1.9506,E1 25.1523,E2 432.4207} C_DIS
LIN {X 97.9014,Y 34.4438,Z 107,A 15.3965,B 24.9278,C -1.9623,E1 25.1501,E2 430.0536} C_DIS
LIN {X 96.7652,Y 37.5201,Z 107,A 17.1463,B 24.9276,C -1.965,E1 25.1484,E2 428.307} C_DIS
LIN {X 95.3664,Y 40.9468,Z 107,A 19.1832,B 24.9272,C -1.9707,E1 25.1462,E2 426.268} C_DIS
LIN {X 93.0488,Y 45.9672,Z 107,A 21.7298,B 24.9281,C -1.9582,E1 25.1432,E2 423.7646} C_DIS
LIN {X 92.0907,Y 47.861,Z 107,A 23.3123,B 24.9266,C -1.9785,E1 25.1411,E2 422.1425} C_DIS
LIN {X 90.5428,Y 50.7254,Z 107,A 25.24,B 24.9258,C -1.9889,E1 25.1385,E2 420.2004} C_DIS
LIN {X 88.4174,Y 54.3479,Z 107,A 27.476,B 24.9256,C -1.9916,E1 25.1353,E2 417.9694} C_DIS
LIN {X 86.2929,Y 57.6619,Z 107,A 29.7023,B 24.925,C -1.9994,E1 25.1319,E2 415.7358} C_DIS
LIN {X 83.738,Y 61.3107,Z 107,A 31.9211,B 24.9253,C -1.9957,E1 25.1283,E2 413.5366} C_DIS
LIN {X 81.7611,Y 63.9254,Z 107,A 34.0052,B 24.9241,C -2.0114,E1 25.1247,E2 411.4252} C_DIS
LIN {X 79.083,Y 67.2082,Z 107,A 36.0544,B 24.9246,C -2.005,E1 25.1211,E2 409.4006} C_DIS
LIN {X 76.9359,Y 69.6581,Z 107,A 37.9732,B 24.9239,C -2.014,E1 25.1175,E2 407.4691} C_DIS
LIN {X 73.5519,Y 73.2211,Z 107,A 40.5685,B 24.9239,C -2.0151,E1 25.1124,E2 404.8824} C_DIS
LIN {X 67.8705,Y 78.517,Z 107,A 44.6165,B 24.9239,C -2.0139,E1 25.1042,E2 400.8535} C_DIS
LIN {X 64.9187,Y 80.9748,Z 107,A 46.9614,B 24.923,C -2.0271,E1 25.0991,E2 398.4865} C_DIS
LIN {X 62.1461,Y 83.1202,Z 107,A 48.737,B 24.9232,C -2.0241,E1 25.0952,E2 396.7244} C_DIS
LIN {X 59.8135,Y 84.8158,Z 107,A 50.5544,B 24.9223,C -2.0359,E1 25.091,E2 394.8854} C_DIS
LIN {X 56.5605,Y 87.019,Z 107,A 52.4961,B 24.9227,C -2.0302,E1 25.0865,E2 392.9635} C_DIS
LIN {X 52.7995,Y 89.3491,Z 107,A 55.0334,B 24.9221,C -2.0378,E1 25.0804,E2 390.4164} C_DIS
LIN {X 49.4243,Y 91.2595,Z 107,A 57.1757,B 24.9219,C -2.0408,E1 25.0752,E2 388.2731} C_DIS
LIN {X 46.2547,Y 92.9063,Z 107,A 59.1375,B 24.9217,C -2.0429,E1 25.0703,E2 386.3117} C_DIS
LIN {X 42.9305,Y 94.4888,Z 107,A 61.2236,B 24.9214,C -2.0475,E1 25.065,E2 384.2202} C_DIS
LIN {X 39.5901,Y 95.9371,Z 107,A 63.1723,B 24.9214,C -2.0472,E1 25.06,E2 382.2768} C_DIS
LIN {X 36.2269,Y 97.2573,Z 107,A 65.3519,B 24.9207,C -2.0565,E1 25.0543,E2 380.08} C_DIS
LIN {X 30.5528,Y 99.1847,Z 107,A 68.3477,B 24.9214,C -2.0468,E1 25.0464,E2 377.1126} C_DIS
LIN {X 27.7714,Y 100.0005,Z 107,A 70.2028,B 24.9206,C -2.058,E1 25.0414,E2 375.2344} C_DIS
LIN {X 24.027,Y 100.9658,Z 107,A 72.1102,B 24.9212,C -2.0503,E1 25.0363,E2 373.348} C_DIS
LIN {X 20.9579,Y 101.6456,Z 107,A 73.8943,B 24.921,C -2.0531,E1 25.0314,E2 371.5596} C_DIS
LIN {X 17.669,Y 102.2695,Z 107,A 75.8791,B 24.9205,C -2.0591,E1 25.0259,E2 369.5627} C_DIS
LIN {X 13.9566,Y 102.8429,Z 107,A 77.7569,B 24.921,C -2.052,E1 25.0208,E2 367.7033} C_DIS
LIN {X 10.8937,Y 103.2104,Z 107,A 79.5962,B 24.9206,C -2.0576,E1 25.0156,E2 365.852} C_DIS
LIN {X 7.7189,Y 103.4977,Z 107,A 81.4311,B 24.9204,C -2.0606,E1 25.0105,E2 364.011} C_DIS
LIN {X 4.1687,Y 103.7003,Z 107,A 83.102,B 24.9213,C -2.0493,E1 25.0059,E2 362.3675} C_DIS
LIN {X 1.4639,Y 103.7743,Z 107,A 84.8971,B 24.9204,C -2.0606,E1 25.0008,E2 360.5457} C_DIS
LIN {X -2.1393,Y 103.7619,Z 107,A 86.8612,B 24.9204,C -2.0592,E1 24.9954,E2 358.585} C_DIS
LIN {X -6.4999,Y 103.5809,Z 107,A 89.0955,B 24.9211,C -2.0516,E1 24.9892,E2 356.368} C_DIS
LIN {X -8.81,Y 103.4105,Z 107,A 90.5702,B 24.9205,C -2.0585,E1 24.985,E2 354.8763} C_DIS
LIN {X -12.6889,Y 103.0069,Z 107,A 92.7449,B 24.9205,C -2.0581,E1 24.979,E2 352.7012} C_DIS
LIN {X -16.2231,Y 102.5085,Z 107,A 94.4446,B 24.9215,C -2.0466,E1 24.9744,E2 351.0275} C_DIS
LIN {X -18.8379,Y 102.0608,Z 107,A 95.9522,B 24.9215,C -2.0471,E1 24.9702,E2 349.5172} C_DIS
LIN {X -21.0553,Y 101.6256,Z 107,A 97.3948,B 24.9209,C -2.0534,E1 24.9662,E2 348.0578} C_DIS
LIN {X -27.3589,Y 100.1131,Z 107,A 100.5309,B 24.9225,C -2.0333,E1 24.9579,E2 344.9651} C_DIS
LIN {X -34.4451,Y 97.9009,Z 107,A 104.9362,B 24.922,C -2.0399,E1 24.9461,E2 340.5364} C_DIS
LIN {X -37.8584,Y 96.6323,Z 107,A 107.0473,B 24.9219,C -2.0409,E1 24.9405,E2 338.4183} C_DIS
LIN {X -40.4838,Y 95.5623,Z 107,A 108.648,B 24.9219,C -2.04,E1 24.9364,E2 336.8162} C_DIS
LIN {X -43.9334,Y 94.0262,Z 107,A 110.6992,B 24.9223,C -2.0356,E1 24.9312,E2 334.7704} C_DIS
Enddeposition()
END
